Yaskawa INFORM job: DEMO_ROOF_SIDE_0625_3PAINT_14.JBI

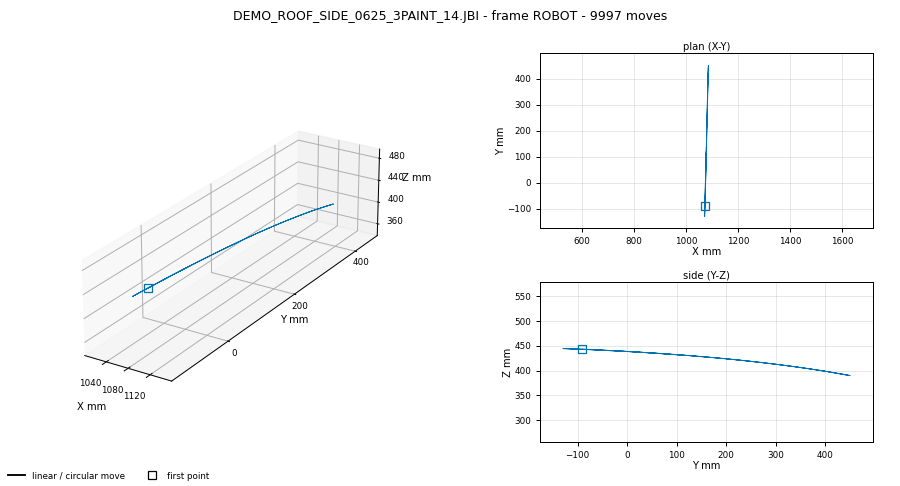
[picture p0: tool path of DEMO_ROOF_SIDE_0625_3PAINT_14.JBI in frame ROBOT, 9997 of 9997 moves have a stored position in this frame; points joined in program order, loops and branches not executed]
/JOB
//NAME DEMO_ROOF_SIDE_0625_3PAINT14
//POS
///NPOS 9997,0,0,0,0,0
///TOOL 0
///USER 0
///POSTYPE ROBOT
///RECTAN
///RCONF 1,0,0,0,0,0,0,0,0,0,0,0,0,0,0,0,0,0,0,0,0,0,0,0
C00000=1074.095,-91.297,443.530,172.904,21.219,153.796
C00001=1074.101,-91.048,443.519,172.905,21.220,153.796
C00002=1074.107,-90.797,443.509,172.907,21.222,153.796
C00003=1074.113,-90.548,443.498,172.908,21.223,153.796
C00004=1074.120,-90.298,443.488,172.910,21.225,153.796
C00005=1074.125,-90.048,443.478,172.911,21.226,153.796
C00006=1074.131,-89.799,443.467,172.913,21.228,153.796
C00007=1074.138,-89.549,443.456,172.914,21.229,153.796
C00008=1074.143,-89.299,443.446,172.916,21.231,153.796
C00009=1074.150,-89.050,443.436,172.917,21.232,153.796
C00010=1074.156,-88.800,443.425,172.919,21.234,153.796
C00011=1074.161,-88.550,443.415,172.921,21.235,153.796
C00012=1074.168,-88.300,443.404,172.922,21.237,153.796
C00013=1074.174,-88.051,443.393,172.924,21.238,153.796
C00014=1074.180,-87.801,443.383,172.925,21.239,153.796
C00015=1074.186,-87.551,443.373,172.927,21.241,153.797
C00016=1074.192,-87.301,443.361,172.928,21.242,153.797
C00017=1074.198,-87.052,443.351,172.930,21.244,153.797
C00018=1074.204,-86.803,443.340,172.931,21.246,153.797
C00019=1074.210,-86.552,443.330,172.933,21.247,153.797
C00020=1074.217,-86.303,443.319,172.934,21.248,153.797
C00021=1074.222,-86.053,443.308,172.936,21.250,153.797
C00022=1074.229,-85.804,443.298,172.937,21.251,153.797
C00023=1074.235,-85.554,443.287,172.939,21.253,153.797
C00024=1074.241,-85.304,443.277,172.941,21.254,153.797
C00025=1074.247,-85.054,443.266,172.942,21.255,153.797
C00026=1074.253,-84.805,443.256,172.943,21.257,153.797
C00027=1074.259,-84.555,443.244,172.945,21.259,153.797
C00028=1074.266,-84.306,443.234,172.947,21.260,153.797
C00029=1074.271,-84.055,443.224,172.948,21.262,153.797
C00030=1074.277,-83.806,443.213,172.950,21.263,153.797
C00031=1074.284,-83.556,443.202,172.951,21.264,153.797
C00032=1074.290,-83.307,443.192,172.953,21.266,153.797
C00033=1074.296,-83.057,443.181,172.954,21.268,153.797
C00034=1074.303,-82.807,443.170,172.956,21.269,153.797
C00035=1074.308,-82.558,443.159,172.957,21.271,153.797
C00036=1074.314,-82.308,443.149,172.959,21.272,153.797
C00037=1074.321,-82.029,443.137,172.961,21.274,153.797
C00038=1074.328,-81.750,443.125,172.962,21.276,153.797
C00039=1074.335,-81.471,443.113,172.964,21.277,153.797
C00040=1074.342,-81.192,443.101,172.965,21.279,153.798
C00041=1074.348,-80.942,443.090,172.967,21.281,153.798
C00042=1074.354,-80.693,443.079,172.968,21.282,153.798
C00043=1074.361,-80.443,443.068,172.971,21.284,153.798
C00044=1074.366,-80.193,443.057,172.972,21.285,153.798
C00045=1074.372,-79.944,443.047,172.974,21.287,153.798
C00046=1074.379,-79.694,443.036,172.975,21.289,153.798
C00047=1074.385,-79.444,443.025,172.977,21.290,153.798
C00048=1074.391,-79.195,443.014,172.978,21.292,153.798
C00049=1074.397,-78.945,443.003,172.980,21.294,153.798
C00050=1074.403,-78.695,442.992,172.981,21.295,153.798
C00051=1074.409,-78.446,442.981,172.983,21.297,153.798
C00052=1074.415,-78.196,442.970,172.984,21.298,153.798
C00053=1074.421,-77.946,442.959,172.986,21.300,153.798
C00054=1074.426,-77.697,442.948,172.987,21.302,153.798
C00055=1074.434,-77.447,442.938,172.989,21.303,153.798
C00056=1074.439,-77.197,442.927,172.990,21.305,153.799
C00057=1074.445,-76.948,442.916,172.992,21.306,153.799
C00058=1074.451,-76.698,442.905,172.993,21.308,153.799
C00059=1074.457,-76.448,442.894,172.995,21.310,153.799
C00060=1074.463,-76.199,442.883,172.996,21.311,153.799
C00061=1074.469,-75.948,442.872,172.997,21.313,153.799
C00062=1074.475,-75.699,442.861,172.999,21.315,153.799
C00063=1074.481,-75.449,442.850,173.001,21.316,153.799
C00064=1074.487,-75.199,442.839,173.002,21.318,153.799
C00065=1074.493,-74.950,442.828,173.003,21.319,153.799
C00066=1074.500,-74.700,442.817,173.005,21.321,153.799
C00067=1074.506,-74.450,442.806,173.006,21.323,153.799
C00068=1074.512,-74.201,442.795,173.008,21.324,153.799
C00069=1074.518,-73.951,442.783,173.009,21.326,153.800
C00070=1074.524,-73.702,442.772,173.011,21.328,153.800
C00071=1074.529,-73.452,442.762,173.012,21.329,153.800
C00072=1074.535,-73.202,442.750,173.014,21.331,153.800
C00073=1074.541,-72.952,442.739,173.015,21.333,153.800
C00074=1074.547,-72.702,442.728,173.016,21.335,153.800
C00075=1074.553,-72.453,442.717,173.019,21.337,153.800
C00076=1074.559,-72.204,442.705,173.020,21.339,153.800
C00077=1074.565,-71.954,442.694,173.022,21.340,153.800
C00078=1074.571,-71.704,442.683,173.023,21.342,153.800
C00079=1074.577,-71.455,442.672,173.025,21.343,153.800
C00080=1074.582,-71.204,442.660,173.026,21.345,153.800
C00081=1074.588,-70.955,442.649,173.027,21.347,153.801
C00082=1074.594,-70.706,442.638,173.029,21.349,153.801
C00083=1074.600,-70.456,442.627,173.030,21.351,153.801
C00084=1074.606,-70.206,442.616,173.032,21.352,153.801
C00085=1074.612,-69.956,442.604,173.033,21.354,153.801
C00086=1074.619,-69.707,442.593,173.035,21.356,153.801
C00087=1074.624,-69.457,442.581,173.036,21.357,153.801
C00088=1074.630,-69.207,442.570,173.037,21.359,153.801
C00089=1074.636,-68.957,442.559,173.039,21.361,153.801
C00090=1074.642,-68.708,442.547,173.040,21.363,153.802
C00091=1074.648,-68.458,442.536,173.042,21.365,153.802
C00092=1074.654,-68.209,442.526,173.043,21.366,153.802
C00093=1074.660,-67.959,442.513,173.045,21.368,153.802
C00094=1074.665,-67.710,442.502,173.046,21.370,153.802
C00095=1074.672,-67.459,442.491,173.048,21.372,153.802
C00096=1074.677,-67.210,442.480,173.050,21.374,153.802
C00097=1074.684,-66.960,442.468,173.051,21.376,153.802
C00098=1074.690,-66.711,442.457,173.053,21.377,153.802
C00099=1074.695,-66.460,442.445,173.054,21.379,153.802
C00100=1074.701,-66.211,442.434,173.055,21.381,153.803
C00101=1074.708,-65.934,442.421,173.057,21.383,153.803
C00102=1074.715,-65.658,442.408,173.058,21.384,153.803
C00103=1074.721,-65.381,442.396,173.060,21.387,153.803
C00104=1074.728,-65.104,442.384,173.062,21.389,153.803
C00105=1074.734,-64.855,442.372,173.063,21.391,153.803
C00106=1074.740,-64.605,442.361,173.065,21.392,153.803
C00107=1074.747,-64.356,442.349,173.066,21.394,153.803
C00108=1074.752,-64.106,442.338,173.067,21.396,153.804
C00109=1074.758,-63.856,442.326,173.069,21.397,153.804
C00110=1074.764,-63.607,442.315,173.070,21.399,153.804
C00111=1074.770,-63.357,442.303,173.072,21.401,153.804
C00112=1074.776,-63.107,442.291,173.073,21.403,153.804
C00113=1074.782,-62.857,442.280,173.075,21.405,153.804
C00114=1074.788,-62.608,442.268,173.077,21.407,153.804
C00115=1074.794,-62.358,442.257,173.078,21.409,153.804
C00116=1074.800,-62.109,442.246,173.080,21.410,153.804
C00117=1074.806,-61.859,442.234,173.081,21.412,153.804
C00118=1074.812,-61.609,442.223,173.082,21.414,153.805
C00119=1074.818,-61.360,442.211,173.084,21.416,153.805
C00120=1074.825,-61.109,442.200,173.085,21.418,153.805
C00121=1074.830,-60.860,442.187,173.087,21.420,153.805
C00122=1074.836,-60.610,442.176,173.088,21.422,153.805
C00123=1074.842,-60.361,442.165,173.090,21.423,153.805
C00124=1074.849,-60.111,442.153,173.091,21.425,153.805
C00125=1074.854,-59.862,442.141,173.092,21.427,153.805
C00126=1074.860,-59.612,442.130,173.094,21.429,153.806
C00127=1074.867,-59.362,442.118,173.095,21.430,153.806
C00128=1074.872,-59.112,442.107,173.097,21.433,153.806
C00129=1074.879,-58.863,442.095,173.099,21.435,153.806
C00130=1074.884,-58.613,442.084,173.100,21.437,153.806
C00131=1074.891,-58.364,442.072,173.102,21.438,153.806
C00132=1074.897,-58.114,442.059,173.103,21.440,153.806
C00133=1074.903,-57.864,442.048,173.104,21.442,153.806
C00134=1074.909,-57.615,442.036,173.106,21.444,153.807
C00135=1074.914,-57.365,442.025,173.107,21.446,153.807
C00136=1074.921,-57.115,442.013,173.109,21.447,153.807
C00137=1074.928,-56.866,442.001,173.110,21.449,153.807
C00138=1074.933,-56.616,441.990,173.111,21.451,153.807
C00139=1074.939,-56.366,441.978,173.113,21.453,153.807
C00140=1074.946,-56.116,441.966,173.114,21.455,153.807
C00141=1074.952,-55.867,441.955,173.117,21.457,153.807
C00142=1074.958,-55.617,441.942,173.118,21.459,153.807
C00143=1074.964,-55.367,441.931,173.119,21.461,153.808
C00144=1074.970,-55.118,441.919,173.121,21.463,153.808
C00145=1074.976,-54.869,441.907,173.122,21.465,153.808
C00146=1074.982,-54.618,441.896,173.124,21.466,153.808
C00147=1074.988,-54.369,441.884,173.125,21.468,153.808
C00148=1074.994,-54.120,441.871,173.126,21.470,153.808
C00149=1075.001,-53.869,441.860,173.128,21.472,153.808
C00150=1075.007,-53.621,441.849,173.129,21.474,153.809
C00151=1075.013,-53.371,441.836,173.130,21.476,153.809
C00152=1075.019,-53.120,441.825,173.132,21.477,153.809
C00153=1075.025,-52.872,441.813,173.134,21.480,153.809
C00154=1075.031,-52.622,441.801,173.135,21.482,153.809
C00155=1075.037,-52.372,441.789,173.137,21.484,153.809
C00156=1075.043,-52.123,441.778,173.138,21.486,153.809
C00157=1075.049,-51.873,441.765,173.140,21.487,153.810
C00158=1075.056,-51.623,441.753,173.141,21.489,153.810
C00159=1075.062,-51.374,441.741,173.142,21.491,153.810
C00160=1075.067,-51.124,441.730,173.144,21.493,153.810
C00161=1075.074,-50.874,441.718,173.145,21.495,153.810
C00162=1075.080,-50.624,441.705,173.147,21.497,153.810
C00163=1075.087,-50.375,441.693,173.148,21.499,153.810
C00164=1075.092,-50.126,441.681,173.150,21.501,153.810
C00165=1075.098,-49.850,441.668,173.152,21.503,153.811
C00166=1075.105,-49.574,441.655,173.153,21.505,153.811
C00167=1075.112,-49.299,441.641,173.154,21.507,153.811
C00168=1075.118,-49.023,441.628,173.156,21.510,153.811
C00169=1075.124,-48.774,441.617,173.158,21.512,153.811
C00170=1075.130,-48.524,441.604,173.159,21.514,153.811
C00171=1075.136,-48.274,441.592,173.160,21.516,153.812
C00172=1075.142,-48.025,441.580,173.162,21.518,153.812
C00173=1075.148,-47.776,441.568,173.163,21.520,153.812
C00174=1075.154,-47.525,441.556,173.164,21.521,153.812
C00175=1075.160,-47.276,441.544,173.166,21.523,153.812
C00176=1075.166,-47.026,441.532,173.168,21.526,153.812
C00177=1075.172,-46.777,441.520,173.169,21.528,153.812
C00178=1075.178,-46.527,441.507,173.171,21.530,153.813
C00179=1075.184,-46.278,441.495,173.172,21.532,153.813
C00180=1075.190,-46.028,441.483,173.173,21.534,153.813
C00181=1075.196,-45.778,441.470,173.175,21.536,153.813
C00182=1075.201,-45.529,441.458,173.176,21.537,153.813
C00183=1075.208,-45.279,441.446,173.178,21.539,153.813
C00184=1075.214,-45.030,441.434,173.179,21.542,153.814
C00185=1075.220,-44.780,441.421,173.181,21.544,153.814
C00186=1075.226,-44.530,441.410,173.182,21.546,153.814
C00187=1075.232,-44.280,441.398,173.184,21.548,153.814
C00188=1075.237,-44.030,441.385,173.185,21.550,153.814
C00189=1075.244,-43.781,441.373,173.186,21.552,153.814
C00190=1075.249,-43.532,441.361,173.188,21.554,153.815
C00191=1075.255,-43.282,441.348,173.189,21.556,153.815
C00192=1075.262,-43.032,441.336,173.190,21.558,153.815
C00193=1075.268,-42.782,441.324,173.192,21.560,153.815
C00194=1075.273,-42.533,441.312,173.193,21.562,153.815
C00195=1075.279,-42.283,441.299,173.195,21.565,153.815
C00196=1075.286,-42.034,441.287,173.197,21.567,153.816
C00197=1075.292,-41.784,441.275,173.198,21.569,153.816
C00198=1075.298,-41.535,441.261,173.199,21.571,153.816
C00199=1075.304,-41.286,441.250,173.201,21.573,153.816
C00200=1075.310,-41.036,441.237,173.202,21.574,153.816
C00201=1075.316,-40.786,441.225,173.203,21.576,153.816
C00202=1075.322,-40.536,441.212,173.205,21.578,153.817
C00203=1075.328,-40.286,441.200,173.206,21.580,153.817
C00204=1075.334,-40.037,441.188,173.208,21.583,153.817
C00205=1075.340,-39.787,441.175,173.209,21.585,153.817
C00206=1075.346,-39.538,441.163,173.211,21.587,153.817
C00207=1075.352,-39.288,441.151,173.212,21.589,153.817
C00208=1075.358,-39.038,441.138,173.214,21.591,153.818
C00209=1075.364,-38.789,441.125,173.215,21.593,153.818
C00210=1075.371,-38.539,441.113,173.216,21.595,153.818
C00211=1075.376,-38.290,441.101,173.217,21.597,153.818
C00212=1075.382,-38.040,441.088,173.219,21.599,153.818
C00213=1075.388,-37.790,441.076,173.221,21.602,153.818
C00214=1075.394,-37.540,441.063,173.222,21.604,153.819
C00215=1075.400,-37.291,441.051,173.224,21.606,153.819
C00216=1075.405,-37.042,441.038,173.225,21.608,153.819
C00217=1075.411,-36.792,441.025,173.226,21.610,153.819
C00218=1075.417,-36.542,441.013,173.228,21.612,153.819
C00219=1075.423,-36.292,441.000,173.229,21.614,153.820
C00220=1075.429,-36.042,440.988,173.230,21.616,153.820
C00221=1075.435,-35.794,440.975,173.232,21.619,153.820
C00222=1075.441,-35.544,440.963,173.234,21.621,153.820
C00223=1075.447,-35.294,440.950,173.235,21.623,153.820
C00224=1075.453,-35.045,440.938,173.236,21.625,153.821
C00225=1075.459,-34.795,440.925,173.238,21.627,153.821
C00226=1075.465,-34.545,440.912,173.239,21.629,153.821
C00227=1075.471,-34.295,440.899,173.240,21.632,153.821
C00228=1075.476,-34.046,440.887,173.242,21.633,153.821
C00229=1075.484,-33.772,440.873,173.244,21.636,153.821
C00230=1075.490,-33.496,440.859,173.245,21.638,153.822
C00231=1075.497,-33.221,440.844,173.246,21.640,153.822
C00232=1075.503,-32.946,440.831,173.248,21.643,153.822
C00233=1075.509,-32.696,440.818,173.250,21.645,153.822
C00234=1075.515,-32.447,440.805,173.251,21.648,153.823
C00235=1075.521,-32.198,440.793,173.252,21.650,153.823
C00236=1075.527,-31.948,440.780,173.254,21.651,153.823
C00237=1075.533,-31.698,440.767,173.255,21.653,153.823
C00238=1075.539,-31.449,440.754,173.257,21.656,153.823
C00239=1075.545,-31.199,440.742,173.258,21.658,153.823
C00240=1075.551,-30.949,440.729,173.260,21.660,153.824
C00241=1075.557,-30.699,440.716,173.261,21.663,153.824
C00242=1075.563,-30.450,440.703,173.262,21.665,153.824
C00243=1075.569,-30.200,440.690,173.264,21.667,153.824
C00244=1075.575,-29.950,440.678,173.265,21.669,153.825
C00245=1075.581,-29.701,440.665,173.266,21.671,153.825
C00246=1075.587,-29.451,440.652,173.269,21.673,153.825
C00247=1075.593,-29.201,440.639,173.270,21.675,153.825
C00248=1075.599,-28.952,440.626,173.271,21.678,153.825
C00249=1075.605,-28.702,440.613,173.272,21.680,153.825
C00250=1075.611,-28.453,440.600,173.274,21.682,153.826
C00251=1075.617,-28.204,440.588,173.275,21.684,153.826
C00252=1075.622,-27.954,440.575,173.276,21.686,153.826
C00253=1075.629,-27.705,440.562,173.278,21.688,153.826
C00254=1075.635,-27.455,440.550,173.280,21.691,153.826
C00255=1075.641,-27.206,440.536,173.281,21.693,153.827
C00256=1075.647,-26.956,440.524,173.282,21.695,153.827
C00257=1075.653,-26.706,440.511,173.284,21.697,153.827
C00258=1075.658,-26.456,440.497,173.285,21.699,153.827
C00259=1075.664,-26.207,440.484,173.286,21.702,153.827
C00260=1075.670,-25.957,440.472,173.288,21.704,153.828
C00261=1075.676,-25.708,440.458,173.290,21.706,153.828
C00262=1075.682,-25.458,440.446,173.291,21.709,153.828
C00263=1075.688,-25.208,440.432,173.292,21.710,153.828
C00264=1075.694,-24.958,440.419,173.294,21.713,153.828
C00265=1075.700,-24.709,440.406,173.295,21.715,153.829
C00266=1075.706,-24.459,440.393,173.296,21.717,153.829
C00267=1075.712,-24.210,440.380,173.297,21.719,153.829
C00268=1075.718,-23.960,440.366,173.300,21.722,153.829
C00269=1075.723,-23.711,440.354,173.301,21.724,153.830
C00270=1075.730,-23.461,440.341,173.302,21.726,153.830
C00271=1075.736,-23.211,440.328,173.303,21.729,153.830
C00272=1075.741,-22.962,440.314,173.305,21.730,153.830
C00273=1075.747,-22.712,440.302,173.306,21.733,153.830
C00274=1075.753,-22.463,440.288,173.307,21.735,153.831
C00275=1075.759,-22.213,440.275,173.308,21.737,153.831
C00276=1075.765,-21.963,440.262,173.311,21.740,153.831
C00277=1075.771,-21.714,440.249,173.312,21.742,153.831
C00278=1075.777,-21.465,440.235,173.313,21.744,153.831
C00279=1075.783,-21.215,440.223,173.315,21.746,153.832
C00280=1075.788,-20.965,440.209,173.316,21.749,153.832
C00281=1075.795,-20.716,440.196,173.317,21.751,153.832
C00282=1075.800,-20.466,440.183,173.318,21.753,153.832
C00283=1075.807,-20.217,440.170,173.321,21.755,153.832
C00284=1075.812,-19.967,440.156,173.322,21.758,153.833
C00285=1075.818,-19.717,440.143,173.323,21.760,153.833
C00286=1075.824,-19.468,440.130,173.324,21.762,153.833
C00287=1075.831,-19.219,440.117,173.326,21.764,153.833
C00288=1075.836,-18.969,440.104,173.327,21.767,153.834
C00289=1075.842,-18.719,440.090,173.328,21.769,153.834
C00290=1075.849,-18.469,440.077,173.330,21.772,153.834
C00291=1075.854,-18.220,440.063,173.332,21.773,153.834
C00292=1075.860,-17.970,440.050,173.333,21.776,153.834
C00293=1075.866,-17.695,440.036,173.334,21.778,153.835
C00294=1075.873,-17.419,440.021,173.336,21.781,153.835
C00295=1075.880,-17.143,440.006,173.337,21.783,153.835
C00296=1075.887,-16.866,439.991,173.339,21.785,153.835
C00297=1075.893,-16.617,439.978,173.341,21.788,153.836
C00298=1075.899,-16.368,439.965,173.342,21.790,153.836
C00299=1075.904,-16.118,439.952,173.343,21.792,153.836
C00300=1075.910,-15.868,439.938,173.345,21.794,153.836
C00301=1075.917,-15.619,439.925,173.346,21.797,153.836
C00302=1075.922,-15.370,439.911,173.347,21.799,153.837
C00303=1075.928,-15.120,439.898,173.349,21.801,153.837
C00304=1075.935,-14.870,439.884,173.351,21.804,153.837
C00305=1075.940,-14.620,439.871,173.352,21.806,153.837
C00306=1075.947,-14.371,439.858,173.353,21.809,153.838
C00307=1075.952,-14.121,439.844,173.354,21.811,153.838
C00308=1075.958,-13.872,439.831,173.356,21.813,153.838
C00309=1075.964,-13.623,439.817,173.357,21.815,153.838
C00310=1075.970,-13.373,439.804,173.359,21.818,153.839
C00311=1075.975,-13.124,439.790,173.360,21.820,153.839
C00312=1075.981,-12.874,439.777,173.362,21.822,153.839
C00313=1075.987,-12.624,439.763,173.363,21.825,153.839
C00314=1075.994,-12.374,439.750,173.364,21.827,153.839
C00315=1075.999,-12.125,439.736,173.365,21.829,153.840
C00316=1076.005,-11.875,439.723,173.367,21.831,153.840
C00317=1076.011,-11.626,439.709,173.369,21.834,153.840
C00318=1076.016,-11.376,439.695,173.370,21.836,153.840
C00319=1076.022,-11.127,439.682,173.371,21.838,153.841
C00320=1076.028,-10.877,439.668,173.373,21.841,153.841
C00321=1076.035,-10.627,439.654,173.374,21.843,153.841
C00322=1076.040,-10.378,439.640,173.375,21.845,153.841
C00323=1076.046,-10.129,439.627,173.377,21.848,153.842
C00324=1076.052,-9.879,439.613,173.379,21.850,153.842
C00325=1076.058,-9.630,439.600,173.380,21.853,153.842
C00326=1076.064,-9.380,439.586,173.381,21.855,153.842
C00327=1076.070,-9.130,439.572,173.382,21.857,153.842
C00328=1076.076,-8.881,439.558,173.383,21.859,153.843
C00329=1076.082,-8.631,439.545,173.386,21.862,153.843
C00330=1076.088,-8.382,439.531,173.387,21.864,153.843
C00331=1076.093,-8.132,439.517,173.388,21.866,153.843
C00332=1076.100,-7.882,439.504,173.389,21.869,153.844
C00333=1076.105,-7.633,439.490,173.391,21.871,153.844
C00334=1076.112,-7.383,439.477,173.392,21.873,153.844
C00335=1076.117,-7.134,439.463,173.393,21.876,153.844
C00336=1076.123,-6.885,439.450,173.395,21.878,153.844
C00337=1076.129,-6.634,439.435,173.397,21.880,153.845
C00338=1076.135,-6.385,439.421,173.398,21.883,153.845
C00339=1076.141,-6.135,439.408,173.399,21.885,153.845
C00340=1076.147,-5.887,439.394,173.400,21.887,153.846
C00341=1076.154,-5.637,439.380,173.402,21.889,153.846
C00342=1076.159,-5.387,439.366,173.404,21.892,153.846
C00343=1076.165,-5.137,439.352,173.405,21.895,153.846
C00344=1076.171,-4.888,439.339,173.406,21.896,153.846
C00345=1076.177,-4.638,439.325,173.408,21.899,153.847
C00346=1076.183,-4.389,439.311,173.409,21.901,153.847
C00347=1076.189,-4.139,439.298,173.410,21.903,153.847
C00348=1076.195,-3.889,439.283,173.412,21.906,153.847
C00349=1076.201,-3.640,439.269,173.414,21.908,153.848
C00350=1076.207,-3.391,439.255,173.415,21.911,153.848
C00351=1076.212,-3.141,439.242,173.416,21.913,153.848
C00352=1076.219,-2.891,439.228,173.417,21.915,153.848
C00353=1076.225,-2.642,439.213,173.419,21.918,153.849
C00354=1076.230,-2.392,439.200,173.421,21.920,153.849
C00355=1076.236,-2.143,439.186,173.422,21.923,153.849
C00356=1076.241,-1.893,439.172,173.423,21.925,153.849
C00357=1076.248,-1.616,439.156,173.424,21.927,153.850
C00358=1076.255,-1.338,439.141,173.426,21.930,153.850
C00359=1076.261,-1.060,439.125,173.428,21.933,153.850
C00360=1076.268,-0.783,439.110,173.429,21.936,153.850
C00361=1076.273,-0.534,439.095,173.431,21.938,153.851
C00362=1076.279,-0.284,439.081,173.432,21.940,153.851
C00363=1076.285,-0.034,439.067,173.433,21.943,153.851
C00364=1076.290,0.215,439.053,173.434,21.945,153.852
C00365=1076.296,0.464,439.038,173.436,21.947,153.852
C00366=1076.302,0.714,439.025,173.438,21.950,153.852
C00367=1076.309,0.964,439.011,173.439,21.953,153.852
C00368=1076.314,1.213,438.996,173.440,21.955,153.853
C00369=1076.320,1.462,438.982,173.442,21.957,153.853
C00370=1076.325,1.712,438.969,173.443,21.960,153.853
C00371=1076.332,1.962,438.954,173.444,21.962,153.853
C00372=1076.337,2.211,438.940,173.446,21.964,153.853
C00373=1076.343,2.461,438.926,173.447,21.967,153.854
C00374=1076.349,2.710,438.911,173.449,21.969,153.854
C00375=1076.355,2.960,438.898,173.450,21.972,153.854
C00376=1076.361,3.209,438.884,173.451,21.974,153.854
C00377=1076.367,3.459,438.869,173.452,21.976,153.855
C00378=1076.373,3.709,438.855,173.454,21.979,153.855
C00379=1076.378,3.957,438.840,173.456,21.981,153.855
C00380=1076.384,4.208,438.826,173.457,21.983,153.855
C00381=1076.390,4.457,438.812,173.458,21.986,153.856
C00382=1076.396,4.706,438.798,173.459,21.988,153.856
C00383=1076.402,4.957,438.784,173.461,21.991,153.856
C00384=1076.408,5.206,438.769,173.463,21.993,153.856
C00385=1076.413,5.455,438.755,173.464,21.996,153.857
C00386=1076.419,5.705,438.740,173.465,21.998,153.857
C00387=1076.425,5.954,438.726,173.466,22.001,153.857
C00388=1076.431,6.203,438.712,173.468,22.002,153.857
C00389=1076.437,6.453,438.698,173.470,22.005,153.858
C00390=1076.443,6.702,438.684,173.471,22.008,153.858
C00391=1076.449,6.952,438.669,173.472,22.010,153.858
C00392=1076.455,7.201,438.655,173.474,22.012,153.858
C00393=1076.461,7.451,438.641,173.475,22.015,153.859
C00394=1076.467,7.701,438.626,173.476,22.017,153.859
C00395=1076.472,7.950,438.612,173.478,22.020,153.859
C00396=1076.479,8.200,438.597,173.480,22.022,153.859
C00397=1076.484,8.449,438.583,173.481,22.024,153.860
C00398=1076.490,8.698,438.569,173.482,22.027,153.860
C00399=1076.496,8.949,438.554,173.483,22.029,153.860
C00400=1076.502,9.198,438.540,173.485,22.032,153.860
C00401=1076.508,9.448,438.526,173.487,22.034,153.861
C00402=1076.514,9.697,438.511,173.488,22.037,153.861
C00403=1076.520,9.947,438.496,173.489,22.039,153.861
C00404=1076.526,10.196,438.482,173.490,22.041,153.862
C00405=1076.532,10.446,438.467,173.492,22.043,153.862
C00406=1076.537,10.695,438.453,173.494,22.046,153.862
C00407=1076.543,10.944,438.439,173.495,22.048,153.862
C00408=1076.550,11.194,438.424,173.496,22.051,153.862
C00409=1076.555,11.444,438.410,173.497,22.053,153.863
C00410=1076.562,11.693,438.395,173.499,22.056,153.863
C00411=1076.567,11.942,438.380,173.501,22.058,153.863
C00412=1076.573,12.192,438.366,173.502,22.060,153.863
C00413=1076.579,12.441,438.352,173.503,22.063,153.864
C00414=1076.586,12.691,438.337,173.505,22.065,153.864
C00415=1076.591,12.941,438.323,173.506,22.067,153.864
C00416=1076.597,13.190,438.308,173.508,22.070,153.864
C00417=1076.603,13.439,438.293,173.509,22.073,153.865
C00418=1076.609,13.690,438.279,173.510,22.075,153.865
C00419=1076.615,13.938,438.265,173.512,22.077,153.865
C00420=1076.621,14.188,438.250,173.513,22.079,153.866
C00421=1076.628,14.468,438.234,173.515,22.082,153.866
C00422=1076.635,14.747,438.217,173.516,22.085,153.866
C00423=1076.641,15.026,438.201,173.518,22.088,153.866
C00424=1076.647,15.306,438.184,173.519,22.090,153.867
C00425=1076.653,15.556,438.169,173.521,22.093,153.867
C00426=1076.659,15.805,438.155,173.522,22.095,153.867
C00427=1076.665,16.054,438.140,173.524,22.098,153.867
C00428=1076.671,16.304,438.125,173.525,22.100,153.868
C00429=1076.677,16.554,438.110,173.526,22.102,153.868
C00430=1076.682,16.803,438.096,173.528,22.105,153.868
C00431=1076.689,17.053,438.081,173.529,22.107,153.869
C00432=1076.695,17.302,438.066,173.531,22.110,153.869
C00433=1076.700,17.552,438.051,173.532,22.113,153.869
C00434=1076.706,17.801,438.037,173.534,22.114,153.869
C00435=1076.712,18.051,438.022,173.535,22.117,153.870
C00436=1076.718,18.300,438.007,173.536,22.119,153.870
C00437=1076.723,18.550,437.992,173.538,22.122,153.870
C00438=1076.729,18.799,437.977,173.539,22.125,153.870
C00439=1076.736,19.048,437.962,173.540,22.127,153.871
C00440=1076.741,19.297,437.948,173.542,22.129,153.871
C00441=1076.747,19.548,437.933,173.543,22.132,153.871
C00442=1076.753,19.797,437.918,173.545,22.134,153.871
C00443=1076.759,20.046,437.903,173.546,22.137,153.872
C00444=1076.765,20.296,437.888,173.548,22.139,153.872
C00445=1076.770,20.545,437.873,173.549,22.141,153.872
C00446=1076.777,20.795,437.858,173.550,22.144,153.872
C00447=1076.783,21.044,437.844,173.552,22.147,153.873
C00448=1076.788,21.294,437.828,173.553,22.149,153.873
C00449=1076.794,21.543,437.814,173.555,22.151,153.873
C00450=1076.800,21.793,437.798,173.556,22.154,153.874
C00451=1076.805,22.042,437.784,173.557,22.156,153.874
C00452=1076.812,22.291,437.769,173.559,22.159,153.874
C00453=1076.817,22.541,437.753,173.560,22.161,153.874
C00454=1076.823,22.790,437.738,173.562,22.164,153.875
C00455=1076.830,23.040,437.723,173.563,22.166,153.875
C00456=1076.835,23.289,437.708,173.564,22.169,153.875
C00457=1076.841,23.539,437.693,173.566,22.171,153.875
C00458=1076.847,23.789,437.678,173.568,22.173,153.876
C00459=1076.852,24.038,437.663,173.569,22.176,153.876
C00460=1076.859,24.288,437.648,173.570,22.178,153.876
C00461=1076.864,24.537,437.633,173.571,22.181,153.876
C00462=1076.870,24.786,437.618,173.573,22.184,153.877
C00463=1076.876,25.036,437.603,173.574,22.186,153.877
C00464=1076.882,25.285,437.588,173.576,22.188,153.877
C00465=1076.888,25.535,437.573,173.577,22.190,153.877
C00466=1076.893,25.784,437.558,173.578,22.193,153.878
C00467=1076.899,26.034,437.543,173.580,22.196,153.878
C00468=1076.905,26.284,437.527,173.582,22.198,153.878
C00469=1076.911,26.533,437.513,173.583,22.200,153.878
C00470=1076.917,26.783,437.498,173.584,22.202,153.879
C00471=1076.923,27.032,437.482,173.585,22.205,153.879
C00472=1076.929,27.281,437.467,173.587,22.208,153.879
C00473=1076.935,27.531,437.452,173.589,22.210,153.880
C00474=1076.940,27.780,437.437,173.590,22.213,153.880
C00475=1076.946,28.030,437.421,173.591,22.215,153.880
C00476=1076.952,28.279,437.406,173.593,22.218,153.880
C00477=1076.958,28.529,437.391,173.595,22.220,153.881
C00478=1076.964,28.778,437.376,173.596,22.222,153.881
C00479=1076.970,29.028,437.360,173.597,22.225,153.881
C00480=1076.976,29.277,437.346,173.598,22.227,153.881
C00481=1076.981,29.527,437.330,173.600,22.230,153.882
C00482=1076.987,29.777,437.314,173.601,22.233,153.882
C00483=1076.993,30.025,437.299,173.603,22.235,153.882
C00484=1076.999,30.275,437.284,173.604,22.237,153.882
C00485=1077.005,30.556,437.267,173.606,22.240,153.883
C00486=1077.012,30.836,437.250,173.607,22.243,153.883
C00487=1077.018,31.117,437.232,173.609,22.246,153.883
C00488=1077.025,31.399,437.215,173.611,22.248,153.884
C00489=1077.031,31.647,437.199,173.612,22.251,153.884
C00490=1077.036,31.897,437.184,173.614,22.253,153.884
C00491=1077.043,32.147,437.169,173.615,22.256,153.885
C00492=1077.048,32.396,437.153,173.616,22.258,153.885
C00493=1077.054,32.624,437.139,173.618,22.260,153.885
C00494=1077.059,32.853,437.125,173.619,22.263,153.885
C00495=1077.064,33.081,437.110,173.620,22.265,153.886
C00496=1077.069,33.310,437.097,173.621,22.267,153.886
C00497=1077.074,33.539,437.083,173.623,22.270,153.886
C00498=1077.080,33.767,437.069,173.624,22.272,153.886
C00499=1077.085,33.995,437.054,173.625,22.274,153.886
C00500=1077.090,34.224,437.040,173.626,22.276,153.887
C00501=1077.097,34.473,437.025,173.629,22.279,153.887
C00502=1077.103,34.723,437.009,173.630,22.281,153.887
C00503=1077.108,34.973,436.993,173.631,22.284,153.888
C00504=1077.114,35.222,436.978,173.632,22.286,153.888
C00505=1077.120,35.471,436.962,173.634,22.289,153.888
C00506=1077.126,35.721,436.947,173.636,22.291,153.888
C00507=1077.132,35.971,436.932,173.637,22.294,153.889
C00508=1077.138,36.219,436.916,173.638,22.296,153.889
C00509=1077.143,36.469,436.900,173.640,22.298,153.889
C00510=1077.150,36.718,436.885,173.642,22.301,153.889
C00511=1077.156,36.968,436.869,173.643,22.303,153.890
C00512=1077.161,37.217,436.854,173.644,22.306,153.890
C00513=1077.167,37.466,436.838,173.645,22.308,153.890
C00514=1077.173,37.716,436.823,173.647,22.311,153.890
C00515=1077.179,37.966,436.806,173.649,22.313,153.891
C00516=1077.184,38.215,436.791,173.650,22.316,153.891
C00517=1077.191,38.464,436.776,173.651,22.318,153.891
C00518=1077.196,38.714,436.760,173.653,22.321,153.891
C00519=1077.202,38.963,436.744,173.654,22.323,153.892
C00520=1077.207,39.213,436.729,173.656,22.326,153.892
C00521=1077.213,39.462,436.712,173.657,22.328,153.892
C00522=1077.219,39.712,436.697,173.658,22.331,153.893
C00523=1077.226,39.961,436.681,173.660,22.333,153.893
C00524=1077.231,40.211,436.666,173.661,22.336,153.893
C00525=1077.237,40.460,436.650,173.663,22.338,153.893
C00526=1077.242,40.710,436.634,173.664,22.340,153.894
C00527=1077.248,40.959,436.618,173.666,22.343,153.894
C00528=1077.254,41.208,436.602,173.667,22.346,153.894
C00529=1077.260,41.458,436.586,173.669,22.348,153.895
C00530=1077.265,41.707,436.570,173.670,22.350,153.895
C00531=1077.271,41.957,436.555,173.672,22.353,153.895
C00532=1077.277,42.206,436.539,173.673,22.356,153.895
C00533=1077.283,42.456,436.523,173.675,22.358,153.896
C00534=1077.289,42.705,436.507,173.676,22.360,153.896
C00535=1077.294,42.954,436.491,173.678,22.363,153.896
C00536=1077.300,43.204,436.476,173.679,22.365,153.896
C00537=1077.306,43.453,436.459,173.680,22.368,153.897
C00538=1077.312,43.703,436.443,173.682,22.370,153.897
C00539=1077.318,43.953,436.428,173.684,22.373,153.897
C00540=1077.323,44.202,436.411,173.685,22.376,153.898
C00541=1077.329,44.451,436.396,173.686,22.378,153.898
C00542=1077.334,44.701,436.380,173.687,22.380,153.898
C00543=1077.340,44.950,436.364,173.689,22.383,153.898
C00544=1077.346,45.199,436.347,173.691,22.386,153.899
C00545=1077.351,45.448,436.332,173.692,22.388,153.899
C00546=1077.357,45.698,436.316,173.693,22.390,153.899
C00547=1077.363,45.947,436.300,173.695,22.393,153.899
C00548=1077.369,46.197,436.284,173.697,22.395,153.900
C00549=1077.376,46.520,436.263,173.698,22.399,153.900
C00550=1077.384,46.843,436.242,173.700,22.402,153.900
C00551=1077.391,47.165,436.222,173.702,22.406,153.901
C00552=1077.398,47.488,436.200,173.703,22.409,153.901
C00553=1077.404,47.737,436.184,173.706,22.411,153.901
C00554=1077.410,47.987,436.169,173.707,22.413,153.902
C00555=1077.416,48.237,436.152,173.708,22.416,153.902
C00556=1077.422,48.486,436.136,173.709,22.418,153.902
C00557=1077.428,48.735,436.120,173.711,22.421,153.903
C00558=1077.433,48.984,436.104,173.713,22.423,153.903
C00559=1077.438,49.234,436.088,173.714,22.426,153.903
C00560=1077.444,49.484,436.071,173.715,22.428,153.903
C00561=1077.450,49.733,436.055,173.717,22.431,153.904
C00562=1077.456,49.982,436.039,173.718,22.434,153.904
C00563=1077.462,50.232,436.023,173.720,22.436,153.904
C00564=1077.468,50.481,436.006,173.721,22.438,153.905
C00565=1077.473,50.731,435.991,173.723,22.441,153.905
C00566=1077.478,50.981,435.974,173.724,22.443,153.905
C00567=1077.484,51.230,435.958,173.726,22.446,153.905
C00568=1077.490,51.479,435.942,173.728,22.448,153.906
C00569=1077.496,51.728,435.926,173.729,22.451,153.906
C00570=1077.502,51.977,435.909,173.730,22.453,153.906
C00571=1077.508,52.227,435.893,173.731,22.456,153.906
C00572=1077.514,52.476,435.877,173.733,22.459,153.907
C00573=1077.519,52.726,435.860,173.735,22.461,153.907
C00574=1077.525,52.975,435.844,173.736,22.463,153.907
C00575=1077.531,53.224,435.827,173.737,22.465,153.907
C00576=1077.537,53.474,435.811,173.739,22.468,153.908
C00577=1077.543,53.723,435.795,173.741,22.471,153.908
C00578=1077.547,53.973,435.779,173.742,22.473,153.908
C00579=1077.553,54.223,435.763,173.743,22.476,153.909
C00580=1077.559,54.472,435.746,173.745,22.478,153.909
C00581=1077.565,54.721,435.730,173.747,22.480,153.909
C00582=1077.571,54.971,435.714,173.748,22.483,153.909
C00583=1077.577,55.220,435.698,173.750,22.486,153.910
C00584=1077.583,55.469,435.680,173.751,22.488,153.910
C00585=1077.589,55.719,435.664,173.752,22.490,153.910
C00586=1077.595,55.968,435.647,173.754,22.493,153.910
C00587=1077.601,56.217,435.631,173.756,22.495,153.911
C00588=1077.606,56.467,435.614,173.757,22.498,153.911
C00589=1077.612,56.716,435.598,173.758,22.500,153.911
C00590=1077.618,56.966,435.582,173.760,22.503,153.911
C00591=1077.624,57.215,435.566,173.762,22.505,153.912
C00592=1077.630,57.464,435.549,173.763,22.508,153.912
C00593=1077.635,57.714,435.533,173.764,22.510,153.912
C00594=1077.641,57.963,435.516,173.767,22.513,153.912
C00595=1077.647,58.213,435.500,173.768,22.515,153.913
C00596=1077.653,58.462,435.484,173.769,22.517,153.913
C00597=1077.658,58.711,435.466,173.770,22.520,153.913
C00598=1077.664,58.960,435.450,173.773,22.522,153.913
C00599=1077.670,59.210,435.434,173.774,22.525,153.914
C00600=1077.676,59.459,435.417,173.775,22.527,153.914
C00601=1077.681,59.709,435.401,173.776,22.529,153.914
C00602=1077.688,59.959,435.384,173.778,22.532,153.915
C00603=1077.694,60.208,435.367,173.780,22.534,153.915
C00604=1077.700,60.457,435.351,173.781,22.537,153.915
C00605=1077.705,60.707,435.334,173.783,22.539,153.915
C00606=1077.711,60.956,435.318,173.784,22.542,153.916
C00607=1077.717,61.205,435.301,173.786,22.544,153.916
C00608=1077.723,61.454,435.284,173.787,22.546,153.916
C00609=1077.729,61.704,435.268,173.789,22.549,153.916
C00610=1077.735,61.953,435.251,173.790,22.551,153.917
C00611=1077.741,62.203,435.235,173.792,22.554,153.917
C00612=1077.746,62.453,435.218,173.794,22.556,153.917
C00613=1077.753,62.732,435.199,173.795,22.559,153.917
C00614=1077.760,63.013,435.181,173.797,22.561,153.918
C00615=1077.766,63.293,435.161,173.798,22.564,153.918
C00616=1077.773,63.574,435.143,173.800,22.567,153.918
C00617=1077.779,63.824,435.127,173.802,22.569,153.918
C00618=1077.785,64.073,435.109,173.803,22.572,153.919
C00619=1077.791,64.323,435.092,173.805,22.574,153.919
C00620=1077.797,64.572,435.076,173.806,22.577,153.919
C00621=1077.803,64.821,435.059,173.808,22.579,153.919
C00622=1077.809,65.071,435.042,173.810,22.582,153.920
C00623=1077.814,65.320,435.025,173.811,22.584,153.920
C00624=1077.820,65.569,435.008,173.812,22.586,153.920
C00625=1077.825,65.819,434.992,173.814,22.589,153.921
C00626=1077.831,66.068,434.975,173.816,22.592,153.921
C00627=1077.837,66.318,434.957,173.817,22.594,153.921
C00628=1077.843,66.567,434.941,173.818,22.596,153.921
C00629=1077.848,66.817,434.924,173.820,22.599,153.922
C00630=1077.855,67.066,434.907,173.822,22.601,153.922
C00631=1077.860,67.315,434.890,173.823,22.604,153.922
C00632=1077.866,67.564,434.873,173.825,22.606,153.922
C00633=1077.871,67.814,434.857,173.826,22.608,153.923
C00634=1077.878,68.063,434.839,173.828,22.611,153.923
C00635=1077.883,68.313,434.822,173.830,22.614,153.923
C00636=1077.889,68.562,434.806,173.831,22.616,153.923
C00637=1077.895,68.811,434.789,173.833,22.618,153.924
C00638=1077.900,69.061,434.772,173.834,22.620,153.924
C00639=1077.906,69.309,434.755,173.836,22.623,153.924
C00640=1077.912,69.560,434.738,173.837,22.626,153.924
C00641=1077.918,69.809,434.720,173.838,22.628,153.925
C00642=1077.924,70.058,434.704,173.841,22.630,153.925
C00643=1077.929,70.307,434.686,173.842,22.633,153.925
C00644=1077.935,70.557,434.670,173.843,22.635,153.925
C00645=1077.941,70.806,434.652,173.845,22.638,153.926
C00646=1077.946,71.056,434.635,173.846,22.641,153.926
C00647=1077.953,71.305,434.618,173.848,22.643,153.926
C00648=1077.958,71.554,434.601,173.850,22.645,153.926
C00649=1077.963,71.803,434.584,173.851,22.648,153.927
C00650=1077.970,72.052,434.567,173.853,22.650,153.927
C00651=1077.976,72.302,434.550,173.854,22.653,153.927
C00652=1077.981,72.552,434.532,173.856,22.655,153.928
C00653=1077.986,72.801,434.515,173.857,22.657,153.928
C00654=1077.993,73.050,434.498,173.859,22.660,153.928
C00655=1077.998,73.299,434.481,173.861,22.662,153.928
C00656=1078.004,73.549,434.463,173.862,22.665,153.929
C00657=1078.010,73.798,434.446,173.863,22.667,153.929
C00658=1078.016,74.047,434.429,173.865,22.670,153.929
C00659=1078.021,74.297,434.412,173.867,22.672,153.929
C00660=1078.027,74.546,434.394,173.868,22.674,153.930
C00661=1078.033,74.795,434.377,173.870,22.677,153.930
C00662=1078.038,75.045,434.360,173.871,22.679,153.930
C00663=1078.044,75.294,434.343,173.873,22.682,153.930
C00664=1078.050,75.544,434.325,173.875,22.684,153.931
C00665=1078.056,75.793,434.308,173.876,22.687,153.931
C00666=1078.062,76.042,434.291,173.877,22.689,153.931
C00667=1078.067,76.291,434.273,173.880,22.692,153.931
C00668=1078.073,76.541,434.256,173.881,22.694,153.932
C00669=1078.079,76.790,434.239,173.882,22.696,153.932
C00670=1078.085,77.039,434.222,173.884,22.699,153.932
C00671=1078.090,77.288,434.204,173.886,22.701,153.932
C00672=1078.096,77.539,434.187,173.887,22.704,153.933
C00673=1078.102,77.788,434.169,173.889,22.706,153.933
C00674=1078.108,78.036,434.152,173.890,22.709,153.933
C00675=1078.114,78.286,434.134,173.892,22.711,153.933
C00676=1078.119,78.536,434.117,173.894,22.714,153.934
C00677=1078.125,78.817,434.097,173.895,22.716,153.934
C00678=1078.132,79.097,434.078,173.897,22.719,153.934
C00679=1078.138,79.377,434.058,173.898,22.721,153.934
C00680=1078.145,79.658,434.039,173.900,22.725,153.935
C00681=1078.150,79.907,434.021,173.902,22.726,153.935
C00682=1078.156,80.156,434.004,173.904,22.729,153.935
C00683=1078.162,80.406,433.986,173.905,22.732,153.936
C00684=1078.168,80.655,433.968,173.906,22.734,153.936
C00685=1078.173,80.904,433.951,173.909,22.737,153.936
C00686=1078.179,81.154,433.933,173.910,22.739,153.936
C00687=1078.184,81.403,433.916,173.911,22.741,153.937
C00688=1078.190,81.652,433.898,173.913,22.744,153.937
C00689=1078.195,81.901,433.881,173.915,22.746,153.937
C00690=1078.202,82.151,433.863,173.916,22.749,153.937
C00691=1078.207,82.400,433.845,173.918,22.751,153.938
C00692=1078.213,82.649,433.828,173.919,22.754,153.938
C00693=1078.219,82.899,433.810,173.922,22.756,153.938
C00694=1078.224,83.148,433.792,173.923,22.759,153.938
C00695=1078.230,83.397,433.775,173.924,22.761,153.939
C00696=1078.236,83.647,433.757,173.926,22.764,153.939
C00697=1078.241,83.896,433.739,173.928,22.766,153.939
C00698=1078.247,84.145,433.722,173.929,22.768,153.939
C00699=1078.253,84.395,433.704,173.931,22.771,153.940
C00700=1078.259,84.644,433.686,173.932,22.773,153.940
C00701=1078.265,84.893,433.668,173.934,22.775,153.940
C00702=1078.270,85.142,433.651,173.936,22.778,153.940
C00703=1078.276,85.391,433.633,173.937,22.780,153.941
C00704=1078.282,85.641,433.615,173.939,22.783,153.941
C00705=1078.287,85.890,433.598,173.941,22.785,153.941
C00706=1078.293,86.140,433.580,173.942,22.787,153.941
C00707=1078.299,86.389,433.562,173.943,22.790,153.942
C00708=1078.305,86.638,433.544,173.945,22.793,153.942
C00709=1078.311,86.888,433.527,173.947,22.794,153.942
C00710=1078.316,87.137,433.509,173.949,22.797,153.942
C00711=1078.322,87.387,433.491,173.950,22.800,153.943
C00712=1078.328,87.636,433.473,173.952,22.802,153.943
C00713=1078.333,87.885,433.456,173.954,22.804,153.943
C00714=1078.339,88.135,433.437,173.955,22.807,153.943
C00715=1078.345,88.383,433.419,173.957,22.809,153.943
C00716=1078.351,88.633,433.401,173.959,22.811,153.944
C00717=1078.356,88.882,433.384,173.960,22.814,153.944
C00718=1078.362,89.132,433.366,173.961,22.816,153.944
C00719=1078.368,89.381,433.348,173.964,22.819,153.944
C00720=1078.374,89.630,433.330,173.965,22.821,153.945
C00721=1078.379,89.879,433.313,173.967,22.823,153.945
C00722=1078.386,90.129,433.294,173.968,22.826,153.945
C00723=1078.391,90.378,433.276,173.970,22.828,153.945
C00724=1078.398,90.627,433.258,173.972,22.830,153.946
C00725=1078.403,90.876,433.241,173.973,22.833,153.946
C00726=1078.408,91.126,433.223,173.974,22.835,153.946
C00727=1078.414,91.375,433.204,173.977,22.837,153.946
C00728=1078.420,91.624,433.186,173.978,22.840,153.947
C00729=1078.425,91.874,433.168,173.980,22.843,153.947
C00730=1078.431,92.123,433.150,173.981,22.845,153.947
C00731=1078.437,92.372,433.132,173.983,22.847,153.947
C00732=1078.443,92.621,433.114,173.985,22.850,153.948
C00733=1078.448,92.871,433.096,173.986,22.852,153.948
C00734=1078.454,93.120,433.078,173.988,22.854,153.948
C00735=1078.459,93.369,433.060,173.990,22.857,153.948
C00736=1078.465,93.619,433.041,173.991,22.859,153.949
C00737=1078.470,93.868,433.024,173.993,22.862,153.949
C00738=1078.477,94.117,433.005,173.995,22.864,153.949
C00739=1078.482,94.366,432.987,173.996,22.866,153.949
C00740=1078.488,94.616,432.969,173.998,22.869,153.949
C00741=1078.494,94.896,432.948,173.999,22.871,153.950
C00742=1078.500,95.177,432.928,174.001,22.874,153.950
C00743=1078.507,95.457,432.907,174.004,22.877,153.950
C00744=1078.513,95.738,432.887,174.006,22.880,153.951
C00745=1078.520,95.987,432.869,174.007,22.882,153.951
C00746=1078.524,96.237,432.851,174.008,22.884,153.951
C00747=1078.531,96.486,432.832,174.011,22.887,153.951
C00748=1078.536,96.735,432.814,174.012,22.889,153.952
C00749=1078.542,96.984,432.795,174.013,22.891,153.952
C00750=1078.547,97.233,432.778,174.016,22.894,153.952
C00751=1078.554,97.483,432.760,174.017,22.896,153.952
C00752=1078.559,97.732,432.741,174.019,22.899,153.953
C00753=1078.565,97.982,432.723,174.020,22.901,153.953
C00754=1078.571,98.231,432.704,174.022,22.903,153.953
C00755=1078.576,98.480,432.686,174.024,22.905,153.953
C00756=1078.582,98.729,432.667,174.025,22.908,153.953
C00757=1078.587,98.979,432.649,174.027,22.911,153.954
C00758=1078.594,99.228,432.631,174.029,22.913,153.954
C00759=1078.599,99.477,432.613,174.030,22.915,153.954
C00760=1078.605,99.726,432.594,174.032,22.917,153.954
C00761=1078.611,99.976,432.576,174.034,22.920,153.955
C00762=1078.617,100.224,432.558,174.036,22.922,153.955
C00763=1078.622,100.474,432.539,174.037,22.924,153.955
C00764=1078.628,100.723,432.521,174.039,22.927,153.955
C00765=1078.633,100.973,432.502,174.041,22.929,153.955
C00766=1078.640,101.222,432.484,174.042,22.931,153.956
C00767=1078.645,101.471,432.465,174.044,22.934,153.956
C00768=1078.651,101.720,432.447,174.046,22.936,153.956
C00769=1078.656,101.969,432.428,174.048,22.939,153.956
C00770=1078.662,102.219,432.410,174.049,22.941,153.957
C00771=1078.668,102.468,432.391,174.051,22.943,153.957
C00772=1078.674,102.717,432.372,174.053,22.946,153.957
C00773=1078.679,102.967,432.354,174.054,22.948,153.957
C00774=1078.684,103.216,432.335,174.056,22.951,153.958
C00775=1078.690,103.465,432.317,174.058,22.953,153.958
C00776=1078.695,103.714,432.298,174.060,22.955,153.958
C00777=1078.702,103.963,432.280,174.061,22.958,153.958
C00778=1078.707,104.213,432.261,174.062,22.960,153.959
C00779=1078.712,104.462,432.242,174.065,22.962,153.959
C00780=1078.719,104.711,432.223,174.066,22.965,153.959
C00781=1078.724,104.960,432.204,174.068,22.967,153.959
C00782=1078.730,105.209,432.187,174.070,22.970,153.960
C00783=1078.736,105.459,432.167,174.071,22.972,153.960
C00784=1078.741,105.708,432.148,174.073,22.974,153.960
C00785=1078.747,105.957,432.131,174.074,22.977,153.960
C00786=1078.752,106.207,432.111,174.077,22.979,153.960
C00787=1078.758,106.456,432.092,174.078,22.981,153.961
C00788=1078.764,106.705,432.074,174.080,22.984,153.961
C00789=1078.769,106.955,432.055,174.082,22.986,153.961
C00790=1078.775,107.203,432.037,174.084,22.989,153.961
C00791=1078.781,107.453,432.018,174.085,22.991,153.962
C00792=1078.787,107.702,431.999,174.086,22.993,153.962
C00793=1078.793,107.951,431.980,174.089,22.995,153.962
C00794=1078.798,108.201,431.962,174.090,22.998,153.962
C00795=1078.803,108.450,431.942,174.092,23.000,153.962
C00796=1078.810,108.699,431.924,174.094,23.002,153.963
C00797=1078.815,108.948,431.905,174.096,23.005,153.963
C00798=1078.821,109.197,431.886,174.097,23.007,153.963
C00799=1078.827,109.446,431.867,174.100,23.009,153.963
C00800=1078.832,109.696,431.849,174.101,23.012,153.964
C00801=1078.838,109.945,431.830,174.102,23.014,153.964
C00802=1078.844,110.194,431.811,174.104,23.016,153.964
C00803=1078.850,110.444,431.792,174.106,23.018,153.964
C00804=1078.855,110.692,431.773,174.108,23.021,153.964
C00805=1078.862,110.973,431.752,174.110,23.024,153.965
C00806=1078.868,111.254,431.730,174.112,23.026,153.965
C00807=1078.875,111.535,431.709,174.114,23.029,153.965
C00808=1078.881,111.815,431.687,174.116,23.031,153.965
C00809=1078.886,112.065,431.669,174.117,23.034,153.966
C00810=1078.893,112.314,431.650,174.120,23.036,153.966
C00811=1078.898,112.563,431.631,174.121,23.038,153.966
C00812=1078.904,112.812,431.612,174.123,23.041,153.966
C00813=1078.909,113.062,431.593,174.124,23.043,153.967
C00814=1078.915,113.311,431.573,174.127,23.045,153.967
C00815=1078.921,113.559,431.555,174.128,23.048,153.967
C00816=1078.926,113.809,431.536,174.130,23.050,153.967
C00817=1078.932,114.058,431.517,174.132,23.052,153.967
C00818=1078.938,114.308,431.497,174.133,23.054,153.968
C00819=1078.943,114.557,431.478,174.135,23.057,153.968
C00820=1078.949,114.805,431.459,174.137,23.059,153.968
C00821=1078.955,115.055,431.439,174.139,23.062,153.968
C00822=1078.960,115.304,431.420,174.140,23.064,153.969
C00823=1078.965,115.553,431.401,174.142,23.066,153.969
C00824=1078.971,115.802,431.382,174.144,23.069,153.969
C00825=1078.977,116.052,431.363,174.146,23.071,153.969
C00826=1078.982,116.301,431.344,174.147,23.073,153.969
C00827=1078.987,116.550,431.325,174.150,23.076,153.970
C00828=1078.993,116.799,431.305,174.151,23.078,153.970
C00829=1078.999,117.049,431.286,174.153,23.081,153.970
C00830=1079.005,117.298,431.267,174.155,23.083,153.970
C00831=1079.010,117.546,431.247,174.157,23.086,153.971
C00832=1079.016,117.796,431.228,174.158,23.087,153.971
C00833=1079.021,118.045,431.209,174.160,23.090,153.971
C00834=1079.027,118.295,431.190,174.162,23.092,153.971
C00835=1079.033,118.544,431.170,174.164,23.095,153.971
C00836=1079.038,118.792,431.151,174.165,23.097,153.972
C00837=1079.044,119.042,431.132,174.168,23.099,153.972
C00838=1079.049,119.291,431.112,174.169,23.101,153.972
C00839=1079.055,119.541,431.093,174.170,23.104,153.972
C00840=1079.061,119.790,431.074,174.173,23.106,153.972
C00841=1079.067,120.039,431.054,174.174,23.108,153.973
C00842=1079.071,120.288,431.034,174.176,23.111,153.973
C00843=1079.077,120.537,431.015,174.178,23.113,153.973
C00844=1079.083,120.787,430.996,174.180,23.115,153.973
C00845=1079.089,121.035,430.976,174.181,23.118,153.974
C00846=1079.094,121.285,430.957,174.183,23.120,153.974
C00847=1079.100,121.534,430.937,174.185,23.122,153.974
C00848=1079.105,121.782,430.918,174.187,23.125,153.974
C00849=1079.111,122.032,430.899,174.188,23.127,153.974
C00850=1079.117,122.281,430.879,174.191,23.129,153.975
C00851=1079.123,122.530,430.859,174.192,23.132,153.975
C00852=1079.128,122.780,430.840,174.194,23.134,153.975
C00853=1079.134,123.029,430.821,174.196,23.136,153.975
C00854=1079.139,123.278,430.800,174.198,23.139,153.975
C00855=1079.145,123.528,430.781,174.200,23.141,153.976
C00856=1079.151,123.777,430.762,174.202,23.143,153.976
C00857=1079.156,124.025,430.742,174.204,23.145,153.976
C00858=1079.162,124.275,430.723,174.205,23.148,153.976
C00859=1079.167,124.524,430.704,174.208,23.150,153.976
C00860=1079.173,124.773,430.684,174.209,23.153,153.977
C00861=1079.179,125.022,430.665,174.211,23.155,153.977
C00862=1079.184,125.271,430.644,174.213,23.157,153.977
C00863=1079.190,125.521,430.625,174.215,23.159,153.977
C00864=1079.196,125.770,430.605,174.216,23.161,153.977
C00865=1079.202,126.019,430.586,174.219,23.164,153.978
C00866=1079.208,126.268,430.566,174.220,23.166,153.978
C00867=1079.213,126.517,430.546,174.222,23.168,153.978
C00868=1079.219,126.766,430.526,174.223,23.171,153.978
C00869=1079.226,127.047,430.505,174.226,23.173,153.978
C00870=1079.231,127.328,430.482,174.228,23.176,153.979
C00871=1079.238,127.608,430.460,174.230,23.178,153.979
C00872=1079.245,127.889,430.437,174.232,23.181,153.979
C00873=1079.250,128.138,430.418,174.234,23.183,153.979
C00874=1079.256,128.387,430.398,174.236,23.185,153.980
C00875=1079.262,128.637,430.379,174.238,23.187,153.980
C00876=1079.268,128.885,430.359,174.240,23.190,153.980
C00877=1079.274,129.135,430.340,174.241,23.192,153.980
C00878=1079.279,129.384,430.319,174.244,23.194,153.980
C00879=1079.285,129.633,430.299,174.245,23.196,153.981
C00880=1079.291,129.882,430.280,174.247,23.199,153.981
C00881=1079.297,130.131,430.260,174.249,23.201,153.981
C00882=1079.302,130.380,430.241,174.251,23.203,153.981
C00883=1079.308,130.630,430.220,174.253,23.206,153.981
C00884=1079.314,130.878,430.200,174.255,23.207,153.981
C00885=1079.319,131.128,430.181,174.257,23.210,153.982
C00886=1079.325,131.377,430.161,174.258,23.212,153.982
C00887=1079.330,131.626,430.140,174.261,23.214,153.982
C00888=1079.336,131.875,430.121,174.262,23.216,153.982
C00889=1079.342,132.124,430.101,174.264,23.218,153.982
C00890=1079.348,132.373,430.081,174.266,23.221,153.983
C00891=1079.353,132.623,430.061,174.268,23.223,153.983
C00892=1079.360,132.872,430.041,174.270,23.226,153.983
C00893=1079.365,133.121,430.020,174.272,23.228,153.983
C00894=1079.371,133.370,430.000,174.274,23.230,153.983
C00895=1079.376,133.620,429.981,174.275,23.232,153.984
C00896=1079.382,133.869,429.961,174.278,23.235,153.984
C00897=1079.388,134.117,429.941,174.279,23.236,153.984
C00898=1079.393,134.367,429.920,174.281,23.239,153.984
C00899=1079.399,134.616,429.901,174.284,23.242,153.984
C00900=1079.404,134.865,429.880,174.285,23.243,153.985
C00901=1079.410,135.114,429.860,174.287,23.246,153.985
C00902=1079.415,135.363,429.840,174.289,23.248,153.985
C00903=1079.421,135.612,429.820,174.291,23.250,153.985
C00904=1079.426,135.862,429.800,174.292,23.253,153.985
C00905=1079.432,136.110,429.780,174.295,23.255,153.986
C00906=1079.438,136.360,429.760,174.297,23.257,153.986
C00907=1079.444,136.608,429.740,174.298,23.260,153.986
C00908=1079.449,136.858,429.719,174.301,23.262,153.986
C00909=1079.455,137.107,429.699,174.302,23.264,153.986
C00910=1079.461,137.356,429.678,174.304,23.266,153.987
C00911=1079.466,137.606,429.659,174.306,23.268,153.987
C00912=1079.472,137.855,429.638,174.308,23.271,153.987
C00913=1079.478,138.103,429.618,174.310,23.273,153.987
C00914=1079.483,138.353,429.598,174.312,23.275,153.987
C00915=1079.489,138.601,429.578,174.314,23.277,153.987
C00916=1079.494,138.851,429.557,174.315,23.280,153.988
C00917=1079.501,139.100,429.537,174.318,23.282,153.988
C00918=1079.506,139.349,429.516,174.320,23.284,153.988
C00919=1079.512,139.598,429.496,174.321,23.286,153.988
C00920=1079.517,139.847,429.476,174.324,23.289,153.988
C00921=1079.523,140.096,429.456,174.325,23.291,153.989
C00922=1079.528,140.345,429.435,174.327,23.293,153.989
C00923=1079.534,140.594,429.415,174.330,23.296,153.989
C00924=1079.540,140.844,429.395,174.331,23.298,153.989
C00925=1079.546,141.093,429.374,174.333,23.300,153.989
C00926=1079.551,141.342,429.353,174.335,23.302,153.990
C00927=1079.557,141.591,429.333,174.337,23.305,153.990
C00928=1079.562,141.840,429.313,174.339,23.307,153.990
C00929=1079.567,142.089,429.292,174.341,23.309,153.990
C00930=1079.573,142.338,429.272,174.343,23.311,153.990
C00931=1079.579,142.588,429.251,174.345,23.313,153.990
C00932=1079.584,142.837,429.231,174.347,23.315,153.991
C00933=1079.591,143.117,429.207,174.349,23.318,153.991
C00934=1079.597,143.398,429.185,174.351,23.321,153.991
C00935=1079.604,143.678,429.161,174.354,23.323,153.991
C00936=1079.610,143.958,429.139,174.356,23.326,153.992
C00937=1079.616,144.208,429.118,174.357,23.328,153.992
C00938=1079.621,144.456,429.097,174.360,23.330,153.992
C00939=1079.626,144.706,429.076,174.362,23.332,153.992
C00940=1079.632,144.954,429.056,174.363,23.335,153.992
C00941=1079.638,145.204,429.035,174.366,23.337,153.992
C00942=1079.644,145.453,429.015,174.368,23.339,153.993
C00943=1079.649,145.702,428.994,174.369,23.341,153.993
C00944=1079.655,145.951,428.974,174.372,23.344,153.993
C00945=1079.660,146.200,428.953,174.373,23.346,153.993
C00946=1079.666,146.450,428.932,174.375,23.348,153.993
C00947=1079.671,146.699,428.912,174.378,23.350,153.993
C00948=1079.678,146.947,428.891,174.379,23.353,153.994
C00949=1079.684,147.197,428.870,174.381,23.355,153.994
C00950=1079.689,147.446,428.849,174.384,23.357,153.994
C00951=1079.694,147.695,428.829,174.385,23.359,153.994
C00952=1079.700,147.943,428.808,174.388,23.361,153.994
C00953=1079.706,148.193,428.787,174.390,23.364,153.995
C00954=1079.712,148.442,428.767,174.391,23.366,153.995
C00955=1079.717,148.691,428.745,174.394,23.368,153.995
C00956=1079.722,148.940,428.725,174.396,23.370,153.995
C00957=1079.728,149.190,428.704,174.397,23.373,153.995
C00958=1079.734,149.438,428.683,174.400,23.375,153.995
C00959=1079.739,149.687,428.662,174.401,23.377,153.996
C00960=1079.746,149.937,428.642,174.403,23.379,153.996
C00961=1079.751,150.185,428.621,174.406,23.382,153.996
C00962=1079.756,150.434,428.600,174.407,23.384,153.996
C00963=1079.762,150.683,428.579,174.409,23.386,153.996
C00964=1079.768,150.933,428.558,174.412,23.388,153.996
C00965=1079.773,151.182,428.537,174.413,23.390,153.997
C00966=1079.779,151.430,428.516,174.415,23.393,153.997
C00967=1079.785,151.680,428.495,174.418,23.395,153.997
C00968=1079.790,151.929,428.474,174.419,23.397,153.997
C00969=1079.795,152.178,428.453,174.422,23.399,153.997
C00970=1079.802,152.427,428.432,174.424,23.402,153.998
C00971=1079.807,152.676,428.411,174.425,23.404,153.998
C00972=1079.812,152.925,428.390,174.428,23.406,153.998
C00973=1079.818,153.174,428.369,174.430,23.408,153.998
C00974=1079.824,153.423,428.348,174.431,23.410,153.998
C00975=1079.829,153.672,428.327,174.434,23.413,153.999
C00976=1079.835,153.921,428.305,174.436,23.415,153.999
C00977=1079.840,154.170,428.285,174.438,23.417,153.999
C00978=1079.846,154.419,428.264,174.440,23.419,153.999
C00979=1079.852,154.669,428.243,174.442,23.422,153.999
C00980=1079.857,154.917,428.221,174.444,23.424,153.999
C00981=1079.863,155.166,428.201,174.446,23.426,154.000
C00982=1079.869,155.415,428.179,174.448,23.428,154.000
C00983=1079.874,155.664,428.158,174.451,23.430,154.000
C00984=1079.880,155.914,428.137,174.452,23.432,154.000
C00985=1079.886,156.162,428.116,174.454,23.435,154.000
C00986=1079.891,156.411,428.095,174.457,23.437,154.000
C00987=1079.896,156.661,428.073,174.458,23.439,154.001
C00988=1079.902,156.909,428.052,174.460,23.441,154.001
C00989=1079.907,157.159,428.031,174.463,23.444,154.001
C00990=1079.913,157.408,428.009,174.465,23.446,154.001
C00991=1079.919,157.656,427.988,174.466,23.448,154.001
C00992=1079.925,157.906,427.967,174.469,23.450,154.001
C00993=1079.930,158.155,427.946,174.471,23.453,154.002
C00994=1079.936,158.403,427.925,174.473,23.454,154.002
C00995=1079.941,158.653,427.903,174.475,23.457,154.002
C00996=1079.947,158.902,427.882,174.477,23.459,154.002
C00997=1079.953,159.182,427.858,174.480,23.462,154.002
C00998=1079.960,159.462,427.834,174.482,23.464,154.003
C00999=1079.966,159.743,427.810,174.484,23.467,154.003
C01000=1079.973,160.023,427.786,174.487,23.469,154.003
C01001=1079.978,160.272,427.765,174.489,23.472,154.003
C01002=1079.984,160.521,427.742,174.490,23.474,154.003
C01003=1079.989,160.770,427.721,174.493,23.476,154.003
C01004=1079.995,161.020,427.700,174.495,23.478,154.004
C01005=1080.001,161.268,427.679,174.497,23.480,154.004
C01006=1080.006,161.517,427.658,174.499,23.482,154.004
C01007=1080.012,161.766,427.635,174.501,23.485,154.004
C01008=1080.017,162.015,427.614,174.503,23.487,154.004
C01009=1080.023,162.264,427.592,174.506,23.489,154.004
C01010=1080.028,162.513,427.571,174.507,23.491,154.005
C01011=1080.033,162.762,427.550,174.509,23.494,154.005
C01012=1080.039,163.011,427.528,174.512,23.496,154.005
C01013=1080.044,163.260,427.506,174.514,23.498,154.005
C01014=1080.050,163.509,427.484,174.515,23.501,154.005
C01015=1080.055,163.758,427.463,174.518,23.503,154.006
C01016=1080.061,164.007,427.441,174.520,23.505,154.006
C01017=1080.066,164.256,427.420,174.523,23.507,154.006
C01018=1080.071,164.505,427.398,174.524,23.510,154.006
C01019=1080.077,164.754,427.376,174.526,23.512,154.006
C01020=1080.082,165.003,427.354,174.529,23.514,154.006
C01021=1080.088,165.252,427.333,174.531,23.516,154.007
C01022=1080.093,165.501,427.311,174.532,23.519,154.007
C01023=1080.099,165.750,427.289,174.535,23.521,154.007
C01024=1080.104,165.999,427.267,174.537,23.523,154.007
C01025=1080.110,166.248,427.246,174.539,23.526,154.007
C01026=1080.115,166.497,427.224,174.541,23.527,154.007
C01027=1080.121,166.746,427.202,174.543,23.530,154.008
C01028=1080.126,166.995,427.180,174.545,23.532,154.008
C01029=1080.132,167.244,427.158,174.548,23.535,154.008
C01030=1080.137,167.493,427.137,174.549,23.536,154.008
C01031=1080.143,167.742,427.115,174.551,23.539,154.008
C01032=1080.148,167.991,427.093,174.554,23.541,154.009
C01033=1080.154,168.240,427.071,174.556,23.544,154.009
C01034=1080.159,168.489,427.050,174.559,23.546,154.009
C01035=1080.165,168.738,427.027,174.560,23.548,154.009
C01036=1080.170,168.986,427.006,174.562,23.550,154.009
C01037=1080.176,169.236,426.983,174.565,23.553,154.009
C01038=1080.182,169.485,426.962,174.567,23.555,154.010
C01039=1080.187,169.734,426.940,174.568,23.557,154.010
C01040=1080.192,169.983,426.918,174.571,23.559,154.010
C01041=1080.198,170.232,426.896,174.573,23.561,154.010
C01042=1080.204,170.481,426.873,174.575,23.563,154.010
C01043=1080.209,170.729,426.852,174.578,23.566,154.010
C01044=1080.215,170.979,426.830,174.579,23.568,154.011
C01045=1080.221,171.228,426.808,174.582,23.570,154.011
C01046=1080.226,171.476,426.786,174.584,23.572,154.011
C01047=1080.231,171.726,426.763,174.586,23.575,154.011
C01048=1080.237,171.974,426.742,174.589,23.577,154.011
C01049=1080.242,172.224,426.720,174.590,23.579,154.011
C01050=1080.249,172.472,426.698,174.592,23.582,154.012
C01051=1080.254,172.721,426.676,174.595,23.584,154.012
C01052=1080.259,172.971,426.654,174.597,23.586,154.012
C01053=1080.265,173.219,426.631,174.599,23.588,154.012
C01054=1080.270,173.468,426.609,174.601,23.590,154.012
C01055=1080.276,173.717,426.588,174.603,23.592,154.012
C01056=1080.282,173.967,426.565,174.606,23.594,154.012
C01057=1080.287,174.215,426.543,174.608,23.597,154.013
C01058=1080.293,174.464,426.521,174.610,23.599,154.013
C01059=1080.299,174.713,426.498,174.613,23.602,154.013
C01060=1080.304,174.962,426.476,174.614,23.604,154.013
C01061=1080.310,175.241,426.452,174.617,23.606,154.013
C01062=1080.317,175.522,426.427,174.620,23.608,154.013
C01063=1080.323,175.802,426.402,174.622,23.611,154.014
C01064=1080.329,176.081,426.376,174.624,23.613,154.014
C01065=1080.336,176.331,426.355,174.627,23.616,154.014
C01066=1080.341,176.579,426.332,174.629,23.618,154.014
C01067=1080.346,176.828,426.310,174.631,23.620,154.014
C01068=1080.352,177.077,426.288,174.633,23.622,154.014
C01069=1080.358,177.326,426.265,174.635,23.624,154.015
C01070=1080.363,177.575,426.243,174.638,23.626,154.015
C01071=1080.369,177.824,426.221,174.640,23.629,154.015
C01072=1080.375,178.073,426.199,174.642,23.631,154.015
C01073=1080.380,178.322,426.176,174.645,23.633,154.015
C01074=1080.386,178.570,426.153,174.647,23.635,154.015
C01075=1080.392,178.820,426.132,174.649,23.637,154.015
C01076=1080.398,179.068,426.109,174.651,23.639,154.016
C01077=1080.403,179.318,426.087,174.653,23.642,154.016
C01078=1080.409,179.567,426.064,174.656,23.644,154.016
C01079=1080.414,179.815,426.042,174.658,23.646,154.016
C01080=1080.420,180.064,426.019,174.660,23.649,154.016
C01081=1080.426,180.313,425.996,174.663,23.651,154.016
C01082=1080.432,180.562,425.975,174.664,23.653,154.017
C01083=1080.438,180.811,425.952,174.667,23.655,154.017
C01084=1080.443,181.061,425.930,174.669,23.657,154.017
C01085=1080.448,181.309,425.907,174.671,23.659,154.017
C01086=1080.455,181.558,425.885,174.674,23.662,154.017
C01087=1080.460,181.807,425.862,174.676,23.664,154.017
C01088=1080.466,182.056,425.840,174.679,23.665,154.017
C01089=1080.472,182.305,425.817,174.681,23.668,154.017
C01090=1080.478,182.554,425.795,174.683,23.670,154.018
C01091=1080.483,182.803,425.772,174.685,23.672,154.018
C01092=1080.489,183.051,425.749,174.687,23.674,154.018
C01093=1080.494,183.300,425.726,174.690,23.676,154.018
C01094=1080.500,183.549,425.705,174.692,23.678,154.018
C01095=1080.506,183.798,425.682,174.694,23.681,154.018
C01096=1080.512,184.047,425.659,174.697,23.683,154.019
C01097=1080.518,184.296,425.636,174.699,23.685,154.019
C01098=1080.524,184.545,425.614,174.702,23.687,154.019
C01099=1080.530,184.794,425.591,174.704,23.690,154.019
C01100=1080.535,185.043,425.568,174.705,23.691,154.019
C01101=1080.540,185.291,425.546,174.708,23.694,154.019
C01102=1080.546,185.540,425.523,174.710,23.696,154.019
C01103=1080.551,185.789,425.499,174.712,23.699,154.020
C01104=1080.557,186.039,425.477,174.715,23.701,154.020
C01105=1080.562,186.288,425.454,174.717,23.703,154.020
C01106=1080.567,186.536,425.432,174.720,23.705,154.020
C01107=1080.573,186.785,425.409,174.722,23.707,154.020
C01108=1080.579,187.034,425.386,174.724,23.710,154.021
C01109=1080.584,187.283,425.362,174.726,23.712,154.021
C01110=1080.590,187.532,425.339,174.729,23.715,154.021
C01111=1080.595,187.781,425.316,174.730,23.716,154.021
C01112=1080.600,188.029,425.294,174.733,23.719,154.021
C01113=1080.606,188.278,425.271,174.735,23.721,154.021
C01114=1080.612,188.527,425.248,174.737,23.724,154.022
C01115=1080.617,188.776,425.224,174.740,23.726,154.022
C01116=1080.622,189.025,425.202,174.742,23.728,154.022
C01117=1080.628,189.274,425.179,174.744,23.730,154.022
C01118=1080.634,189.523,425.156,174.747,23.732,154.022
C01119=1080.640,189.771,425.133,174.749,23.735,154.022
C01120=1080.644,190.020,425.109,174.752,23.737,154.022
C01121=1080.650,190.269,425.086,174.754,23.740,154.023
C01122=1080.656,190.518,425.063,174.756,23.742,154.023
C01123=1080.661,190.767,425.040,174.759,23.744,154.023
C01124=1080.666,191.016,425.017,174.761,23.746,154.023
C01125=1080.673,191.295,424.991,174.763,23.748,154.023
C01126=1080.679,191.575,424.965,174.766,23.751,154.023
C01127=1080.685,191.855,424.939,174.769,23.754,154.024
C01128=1080.692,192.134,424.914,174.771,23.757,154.024
C01129=1080.697,192.383,424.891,174.773,23.759,154.024
C01130=1080.702,192.632,424.867,174.776,23.761,154.024
C01131=1080.708,192.881,424.843,174.778,23.763,154.024
C01132=1080.714,193.129,424.820,174.781,23.765,154.024
C01133=1080.720,193.378,424.797,174.783,23.768,154.025
C01134=1080.725,193.628,424.774,174.785,23.770,154.025
C01135=1080.731,193.877,424.751,174.788,23.772,154.025
C01136=1080.736,194.125,424.728,174.790,23.774,154.025
C01137=1080.742,194.374,424.704,174.793,23.776,154.025
C01138=1080.747,194.623,424.681,174.795,23.779,154.025
C01139=1080.753,194.872,424.658,174.797,23.781,154.026
C01140=1080.759,195.121,424.635,174.800,23.784,154.026
C01141=1080.764,195.369,424.611,174.802,23.786,154.026
C01142=1080.770,195.618,424.588,174.804,23.788,154.026
C01143=1080.775,195.867,424.565,174.807,23.790,154.026
C01144=1080.781,196.116,424.541,174.809,23.792,154.026
C01145=1080.787,196.365,424.518,174.811,23.795,154.026
C01146=1080.792,196.613,424.495,174.814,23.797,154.027
C01147=1080.797,196.863,424.471,174.816,23.799,154.027
C01148=1080.803,197.111,424.447,174.819,23.801,154.027
C01149=1080.809,197.360,424.425,174.821,23.803,154.027
C01150=1080.814,197.608,424.400,174.823,23.806,154.027
C01151=1080.820,197.857,424.377,174.826,23.808,154.027
C01152=1080.826,198.107,424.354,174.828,23.810,154.027
C01153=1080.832,198.355,424.330,174.831,23.812,154.028
C01154=1080.837,198.604,424.307,174.833,23.815,154.028
C01155=1080.843,198.853,424.284,174.835,23.817,154.028
C01156=1080.848,199.102,424.260,174.838,23.819,154.028
C01157=1080.854,199.351,424.237,174.840,23.822,154.028
C01158=1080.860,199.599,424.213,174.842,23.824,154.028
C01159=1080.865,199.848,424.189,174.845,23.826,154.029
C01160=1080.872,200.097,424.165,174.847,23.828,154.029
C01161=1080.878,200.346,424.142,174.850,23.830,154.029
C01162=1080.883,200.595,424.118,174.852,23.833,154.029
C01163=1080.889,200.844,424.095,174.854,23.835,154.029
C01164=1080.894,201.092,424.071,174.857,23.837,154.029
C01165=1080.900,201.341,424.048,174.859,23.839,154.029
C01166=1080.906,201.590,424.024,174.861,23.842,154.030
C01167=1080.911,201.839,424.001,174.864,23.844,154.030
C01168=1080.917,202.088,423.977,174.866,23.846,154.030
C01169=1080.922,202.337,423.953,174.869,23.848,154.030
C01170=1080.928,202.585,423.930,174.871,23.850,154.030
C01171=1080.934,202.834,423.905,174.873,23.853,154.030
C01172=1080.940,203.083,423.882,174.876,23.855,154.030
C01173=1080.945,203.332,423.858,174.878,23.857,154.031
C01174=1080.951,203.580,423.834,174.880,23.860,154.031
C01175=1080.956,203.829,423.811,174.883,23.862,154.031
C01176=1080.962,204.078,423.786,174.885,23.864,154.031
C01177=1080.967,204.327,423.763,174.889,23.867,154.031
C01178=1080.973,204.576,423.739,174.891,23.869,154.031
C01179=1080.979,204.825,423.715,174.893,23.871,154.032
C01180=1080.985,205.073,423.691,174.896,23.873,154.032
C01181=1080.990,205.322,423.667,174.898,23.876,154.032
C01182=1080.995,205.571,423.643,174.900,23.878,154.032
C01183=1081.001,205.819,423.619,174.903,23.880,154.032
C01184=1081.006,206.069,423.596,174.905,23.883,154.032
C01185=1081.012,206.318,423.571,174.907,23.885,154.033
C01186=1081.018,206.566,423.548,174.910,23.887,154.033
C01187=1081.023,206.814,423.523,174.912,23.889,154.033
C01188=1081.029,207.064,423.499,174.915,23.891,154.033
C01189=1081.052,208.096,423.400,175.012,23.943,154.031
C01190=1081.061,208.494,423.360,175.016,23.948,154.032
C01191=1081.071,208.891,423.321,175.019,23.954,154.032
C01192=1081.080,209.288,423.282,175.023,23.959,154.033
C01193=1081.089,209.686,423.243,175.027,23.964,154.034
C01194=1081.094,209.934,423.219,175.029,23.968,154.034
C01195=1081.100,210.183,423.193,175.032,23.971,154.034
C01196=1081.106,210.432,423.169,175.034,23.974,154.035
C01197=1081.111,210.681,423.144,175.036,23.977,154.035
C01198=1081.117,210.929,423.119,175.039,23.980,154.035
C01199=1081.123,211.178,423.095,175.041,23.984,154.036
C01200=1081.128,211.427,423.071,175.043,23.987,154.036
C01201=1081.134,211.676,423.045,175.045,23.990,154.037
C01202=1081.140,211.924,423.021,175.048,23.994,154.037
C01203=1081.145,212.174,422.996,175.050,23.996,154.037
C01204=1081.151,212.422,422.971,175.052,24.000,154.038
C01205=1081.156,212.671,422.946,175.055,24.003,154.038
C01206=1081.162,212.919,422.921,175.057,24.007,154.038
C01207=1081.168,213.168,422.897,175.060,24.010,154.039
C01208=1081.174,213.416,422.872,175.062,24.013,154.039
C01209=1081.179,213.666,422.847,175.065,24.017,154.040
C01210=1081.185,213.914,422.823,175.067,24.020,154.040
C01211=1081.190,214.163,422.797,175.069,24.023,154.040
C01212=1081.195,214.412,422.773,175.071,24.026,154.041
C01213=1081.202,214.660,422.747,175.074,24.029,154.041
C01214=1081.208,214.909,422.722,175.076,24.033,154.042
C01215=1081.213,215.158,422.698,175.078,24.036,154.042
C01216=1081.219,215.407,422.672,175.081,24.039,154.042
C01217=1081.224,215.655,422.647,175.083,24.043,154.043
C01218=1081.230,215.904,422.622,175.085,24.046,154.043
C01219=1081.235,216.152,422.598,175.087,24.049,154.044
C01220=1081.242,216.401,422.572,175.091,24.052,154.044
C01221=1081.247,216.649,422.547,175.093,24.055,154.044
C01222=1081.252,216.899,422.522,175.095,24.059,154.045
C01223=1081.259,217.147,422.497,175.098,24.062,154.045
C01224=1081.264,217.396,422.473,175.100,24.065,154.045
C01225=1081.269,217.645,422.447,175.102,24.069,154.046
C01226=1081.276,217.894,422.421,175.104,24.072,154.046
C01227=1081.281,218.142,422.397,175.107,24.075,154.046
C01228=1081.287,218.391,422.372,175.109,24.078,154.047
C01229=1081.292,218.639,422.346,175.111,24.081,154.047
C01230=1081.298,218.888,422.321,175.114,24.085,154.048
C01231=1081.304,219.137,422.296,175.116,24.088,154.048
C01232=1081.309,219.385,422.271,175.119,24.091,154.048
C01233=1081.315,219.634,422.245,175.121,24.094,154.049
C01234=1081.321,219.883,422.220,175.124,24.098,154.049
C01235=1081.327,220.131,422.196,175.126,24.101,154.050
C01236=1081.332,220.380,422.170,175.128,24.104,154.050
C01237=1081.338,220.629,422.145,175.131,24.108,154.050
C01238=1081.344,220.877,422.120,175.133,24.110,154.051
C01239=1081.349,221.126,422.094,175.135,24.114,154.051
C01240=1081.356,221.375,422.068,175.138,24.117,154.051
C01241=1081.362,221.624,422.044,175.140,24.121,154.052
C01242=1081.370,222.025,422.002,175.144,24.126,154.052
C01243=1081.380,222.426,421.961,175.148,24.131,154.053
C01244=1081.388,222.828,421.920,175.152,24.136,154.054
C01245=1081.398,223.229,421.879,175.155,24.141,154.054
C01246=1081.403,223.478,421.854,175.158,24.145,154.055
C01247=1081.409,223.727,421.828,175.161,24.148,154.055
C01248=1081.414,223.976,421.802,175.163,24.151,154.056
C01249=1081.420,224.224,421.778,175.166,24.155,154.056
C01250=1081.425,224.473,421.752,175.168,24.158,154.056
C01251=1081.432,224.721,421.726,175.170,24.161,154.057
C01252=1081.437,224.970,421.700,175.173,24.165,154.057
C01253=1081.442,225.219,421.675,175.175,24.168,154.057
C01254=1081.448,225.467,421.649,175.177,24.171,154.058
C01255=1081.454,225.716,421.623,175.180,24.175,154.058
C01256=1081.460,225.964,421.597,175.182,24.177,154.058
C01257=1081.465,226.213,421.572,175.185,24.181,154.059
C01258=1081.471,226.461,421.547,175.188,24.184,154.059
C01259=1081.477,226.710,421.521,175.190,24.187,154.060
C01260=1081.483,226.959,421.495,175.193,24.191,154.060
C01261=1081.488,227.208,421.469,175.195,24.194,154.060
C01262=1081.494,227.457,421.443,175.197,24.197,154.061
C01263=1081.500,227.704,421.418,175.200,24.200,154.061
C01264=1081.505,227.953,421.392,175.202,24.204,154.062
C01265=1081.511,228.202,421.366,175.204,24.207,154.062
C01266=1081.517,228.451,421.340,175.207,24.210,154.062
C01267=1081.522,228.700,421.315,175.209,24.214,154.063
C01268=1081.529,228.948,421.289,175.211,24.217,154.063
C01269=1081.534,229.196,421.263,175.215,24.220,154.063
C01270=1081.539,229.445,421.237,175.217,24.223,154.064
C01271=1081.545,229.694,421.212,175.220,24.227,154.064
C01272=1081.551,229.942,421.185,175.222,24.230,154.065
C01273=1081.557,230.191,421.160,175.224,24.233,154.065
C01274=1081.563,230.440,421.134,175.227,24.236,154.065
C01275=1081.569,230.688,421.107,175.229,24.239,154.066
C01276=1081.573,230.936,421.082,175.231,24.243,154.066
C01277=1081.580,231.185,421.056,175.234,24.246,154.066
C01278=1081.585,231.433,421.030,175.236,24.249,154.067
C01279=1081.591,231.682,421.004,175.239,24.253,154.067
C01280=1081.596,231.931,420.978,175.242,24.256,154.068
C01281=1081.602,232.180,420.951,175.244,24.259,154.068
C01282=1081.608,232.429,420.925,175.247,24.263,154.068
C01283=1081.614,232.677,420.899,175.249,24.266,154.069
C01284=1081.620,232.926,420.873,175.251,24.269,154.069
C01285=1081.624,233.174,420.848,175.254,24.272,154.069
C01286=1081.630,233.422,420.821,175.256,24.276,154.070
C01287=1081.636,233.671,420.795,175.259,24.279,154.070
C01288=1081.641,233.920,420.768,175.261,24.282,154.071
C01289=1081.648,234.168,420.743,175.263,24.286,154.071
C01290=1081.653,234.417,420.716,175.266,24.289,154.071
C01291=1081.659,234.666,420.690,175.268,24.292,154.072
C01292=1081.665,234.914,420.664,175.272,24.295,154.072
C01293=1081.670,235.163,420.638,175.274,24.299,154.073
C01294=1081.679,235.556,420.596,175.277,24.304,154.073
C01295=1081.687,235.949,420.554,175.282,24.309,154.074
C01296=1081.697,236.342,420.513,175.285,24.314,154.074
C01297=1081.706,236.735,420.471,175.290,24.320,154.075
C01298=1081.712,236.983,420.445,175.292,24.323,154.075
C01299=1081.717,237.231,420.418,175.294,24.326,154.076
C01300=1081.723,237.480,420.392,175.297,24.330,154.076
C01301=1081.729,237.729,420.365,175.299,24.333,154.077
C01302=1081.734,237.977,420.339,175.302,24.336,154.077
C01303=1081.740,238.226,420.313,175.305,24.339,154.077
C01304=1081.746,238.474,420.286,175.308,24.343,154.078
C01305=1081.751,238.723,420.259,175.310,24.346,154.078
C01306=1081.757,238.971,420.233,175.312,24.349,154.079
C01307=1081.763,239.220,420.207,175.315,24.353,154.079
C01308=1081.768,239.468,420.180,175.317,24.356,154.079
C01309=1081.774,239.717,420.154,175.320,24.359,154.080
C01310=1081.780,239.965,420.127,175.322,24.362,154.080
C01311=1081.786,240.215,420.101,175.325,24.366,154.080
C01312=1081.792,240.463,420.074,175.327,24.369,154.081
C01313=1081.798,240.712,420.047,175.330,24.372,154.081
C01314=1081.803,240.960,420.021,175.333,24.376,154.082
C01315=1081.809,241.208,419.994,175.335,24.379,154.082
C01316=1081.814,241.457,419.967,175.338,24.382,154.082
C01317=1081.820,241.705,419.940,175.340,24.386,154.083
C01318=1081.826,241.954,419.914,175.343,24.389,154.083
C01319=1081.831,242.203,419.888,175.345,24.392,154.083
C01320=1081.837,242.451,419.861,175.348,24.395,154.084
C01321=1081.843,242.700,419.834,175.350,24.399,154.084
C01322=1081.849,242.948,419.807,175.353,24.402,154.085
C01323=1081.855,243.197,419.781,175.355,24.405,154.085
C01324=1081.860,243.446,419.753,175.358,24.408,154.085
C01325=1081.866,243.694,419.727,175.361,24.412,154.086
C01326=1081.871,243.942,419.700,175.363,24.415,154.086
C01327=1081.876,244.191,419.673,175.366,24.419,154.087
C01328=1081.882,244.439,419.646,175.368,24.422,154.087
C01329=1081.888,244.688,419.620,175.371,24.426,154.087
C01330=1081.894,244.937,419.593,175.373,24.429,154.088
C01331=1081.900,245.185,419.565,175.376,24.432,154.088
C01332=1081.905,245.433,419.538,175.378,24.435,154.089
C01333=1081.911,245.681,419.511,175.381,24.439,154.089
C01334=1081.916,245.930,419.484,175.383,24.442,154.089
C01335=1081.922,246.178,419.457,175.386,24.445,154.090
C01336=1081.928,246.427,419.431,175.389,24.448,154.090
C01337=1081.933,246.676,419.403,175.392,24.452,154.091
C01338=1081.939,246.925,419.376,175.394,24.455,154.091
C01339=1081.945,247.172,419.349,175.397,24.459,154.091
C01340=1081.950,247.421,419.322,175.399,24.462,154.092
C01341=1081.956,247.669,419.295,175.402,24.465,154.092
C01342=1081.961,247.918,419.268,175.404,24.469,154.093
C01343=1081.968,248.166,419.240,175.407,24.472,154.093
C01344=1081.973,248.415,419.213,175.409,24.475,154.093
C01345=1081.979,248.663,419.186,175.411,24.479,154.094
C01346=1081.987,249.050,419.143,175.416,24.484,154.094
C01347=1081.995,249.436,419.102,175.419,24.489,154.095
C01348=1082.005,249.822,419.059,175.424,24.495,154.096
C01349=1082.013,250.208,419.017,175.428,24.500,154.096
C01350=1082.019,250.457,418.989,175.431,24.503,154.097
C01351=1082.025,250.705,418.962,175.433,24.506,154.097
C01352=1082.030,250.954,418.934,175.436,24.510,154.097
C01353=1082.036,251.202,418.908,175.438,24.513,154.098
C01354=1082.042,251.451,418.880,175.441,24.517,154.098
C01355=1082.047,251.699,418.853,175.443,24.520,154.099
C01356=1082.053,251.947,418.825,175.446,24.523,154.099
C01357=1082.058,252.196,418.798,175.448,24.527,154.099
C01358=1082.064,252.444,418.770,175.451,24.530,154.100
C01359=1082.070,252.693,418.743,175.454,24.533,154.100
C01360=1082.075,252.941,418.716,175.457,24.537,154.101
C01361=1082.081,253.189,418.688,175.459,24.540,154.101
C01362=1082.087,253.438,418.660,175.462,24.544,154.102
C01363=1082.092,253.686,418.633,175.464,24.547,154.102
C01364=1082.098,253.934,418.605,175.467,24.550,154.102
C01365=1082.104,254.183,418.578,175.470,24.554,154.103
C01366=1082.109,254.432,418.550,175.472,24.557,154.103
C01367=1082.114,254.680,418.523,175.475,24.560,154.103
C01368=1082.121,254.929,418.495,175.477,24.564,154.104
C01369=1082.126,255.177,418.467,175.480,24.567,154.104
C01370=1082.132,255.425,418.440,175.482,24.570,154.105
C01371=1082.138,255.674,418.412,175.486,24.574,154.105
C01372=1082.144,255.922,418.384,175.488,24.577,154.105
C01373=1082.149,256.171,418.357,175.491,24.581,154.106
C01374=1082.155,256.419,418.329,175.493,24.584,154.106
C01375=1082.161,256.667,418.301,175.496,24.587,154.107
C01376=1082.166,256.916,418.274,175.498,24.590,154.107
C01377=1082.172,257.164,418.246,175.501,24.594,154.107
C01378=1082.178,257.413,418.218,175.504,24.598,154.108
C01379=1082.184,257.661,418.190,175.506,24.601,154.108
C01380=1082.189,257.909,418.163,175.509,24.604,154.109
C01381=1082.195,258.158,418.135,175.511,24.607,154.109
C01382=1082.201,258.406,418.107,175.515,24.611,154.109
C01383=1082.207,258.655,418.079,175.517,24.614,154.110
C01384=1082.213,258.903,418.051,175.520,24.618,154.110
C01385=1082.218,259.152,418.024,175.523,24.621,154.111
C01386=1082.224,259.400,417.997,175.525,24.624,154.111
C01387=1082.230,259.648,417.968,175.528,24.628,154.111
C01388=1082.236,259.896,417.940,175.530,24.631,154.112
C01389=1082.242,260.145,417.912,175.533,24.635,154.112
C01390=1082.248,260.393,417.885,175.535,24.638,154.113
C01391=1082.254,260.642,417.856,175.538,24.641,154.113
C01392=1082.259,260.890,417.828,175.541,24.645,154.113
C01393=1082.265,261.139,417.800,175.544,24.648,154.114
C01394=1082.271,261.386,417.773,175.547,24.652,154.114
C01395=1082.277,261.635,417.744,175.549,24.655,154.115
C01396=1082.282,261.883,417.716,175.552,24.658,154.115
C01397=1082.288,262.132,417.688,175.554,24.661,154.115
C01398=1082.297,262.515,417.645,175.559,24.666,154.116
C01399=1082.306,262.899,417.602,175.563,24.672,154.117
C01400=1082.315,263.282,417.559,175.567,24.677,154.117
C01401=1082.325,263.666,417.515,175.571,24.682,154.118
C01402=1082.330,263.914,417.488,175.574,24.685,154.118
C01403=1082.336,264.162,417.458,175.577,24.689,154.119
C01404=1082.342,264.410,417.431,175.579,24.692,154.119
C01405=1082.348,264.659,417.402,175.582,24.696,154.119
C01406=1082.353,264.907,417.374,175.585,24.699,154.120
C01407=1082.359,265.156,417.346,175.587,24.702,154.120
C01408=1082.364,265.404,417.318,175.590,24.706,154.121
C01409=1082.370,265.652,417.289,175.592,24.709,154.121
C01410=1082.376,265.901,417.261,175.595,24.712,154.121
C01411=1082.382,266.149,417.233,175.598,24.716,154.122
C01412=1082.388,266.397,417.204,175.600,24.720,154.122
C01413=1082.393,266.645,417.176,175.603,24.723,154.123
C01414=1082.399,266.894,417.147,175.606,24.726,154.123
C01415=1082.405,267.143,417.118,175.609,24.730,154.124
C01416=1082.410,267.391,417.090,175.612,24.733,154.124
C01417=1082.416,267.639,417.061,175.614,24.736,154.124
C01418=1082.421,267.887,417.033,175.617,24.740,154.125
C01419=1082.427,268.136,417.005,175.620,24.744,154.125
C01420=1082.434,268.384,416.976,175.622,24.747,154.126
C01421=1082.439,268.632,416.948,175.625,24.751,154.126
C01422=1082.445,268.880,416.919,175.627,24.754,154.127
C01423=1082.451,269.129,416.891,175.630,24.757,154.127
C01424=1082.456,269.377,416.862,175.633,24.761,154.127
C01425=1082.462,269.625,416.833,175.636,24.764,154.128
C01426=1082.467,269.873,416.805,175.639,24.768,154.128
C01427=1082.474,270.121,416.776,175.642,24.771,154.128
C01428=1082.480,270.370,416.748,175.644,24.775,154.129
C01429=1082.484,270.618,416.719,175.647,24.778,154.129
C01430=1082.490,270.867,416.690,175.650,24.782,154.130
C01431=1082.497,271.115,416.661,175.652,24.785,154.130
C01432=1082.502,271.363,416.633,175.655,24.788,154.131
C01433=1082.508,271.611,416.604,175.658,24.792,154.131
C01434=1082.513,271.860,416.575,175.660,24.796,154.132
C01435=1082.520,272.108,416.546,175.663,24.799,154.132
C01436=1082.525,272.356,416.518,175.665,24.802,154.132
C01437=1082.531,272.605,416.489,175.669,24.806,154.133
C01438=1082.537,272.853,416.460,175.672,24.809,154.133
C01439=1082.542,273.101,416.432,175.674,24.812,154.134
C01440=1082.548,273.349,416.403,175.677,24.816,154.134
C01441=1082.554,273.597,416.373,175.680,24.820,154.135
C01442=1082.560,273.846,416.345,175.682,24.823,154.135
C01443=1082.565,274.094,416.316,175.685,24.827,154.135
C01444=1082.571,274.342,416.286,175.688,24.830,154.136
C01445=1082.577,274.591,416.258,175.690,24.834,154.136
C01446=1082.582,274.839,416.229,175.693,24.837,154.137
C01447=1082.588,275.087,416.200,175.696,24.841,154.137
C01448=1082.594,275.335,416.171,175.698,24.844,154.137
C01449=1082.600,275.584,416.142,175.701,24.848,154.138
C01450=1082.609,275.970,416.096,175.706,24.853,154.139
C01451=1082.618,276.356,416.051,175.710,24.859,154.139
C01452=1082.626,276.743,416.006,175.714,24.864,154.140
C01453=1082.636,277.129,415.961,175.719,24.870,154.141
C01454=1082.641,277.377,415.931,175.722,24.873,154.141
C01455=1082.647,277.625,415.902,175.724,24.877,154.142
C01456=1082.652,277.874,415.873,175.727,24.880,154.142
C01457=1082.659,278.122,415.844,175.730,24.884,154.142
C01458=1082.664,278.370,415.814,175.733,24.887,154.143
C01459=1082.670,278.618,415.785,175.735,24.891,154.143
C01460=1082.675,278.866,415.756,175.738,24.894,154.144
C01461=1082.682,279.114,415.727,175.741,24.898,154.144
C01462=1082.687,279.363,415.697,175.743,24.902,154.145
C01463=1082.693,279.611,415.668,175.746,24.905,154.145
C01464=1082.699,279.859,415.638,175.749,24.909,154.145
C01465=1082.705,280.107,415.609,175.752,24.912,154.146
C01466=1082.710,280.355,415.580,175.755,24.916,154.146
C01467=1082.715,280.603,415.550,175.758,24.919,154.147
C01468=1082.722,280.852,415.521,175.761,24.923,154.147
C01469=1082.727,281.100,415.492,175.763,24.926,154.148
C01470=1082.733,281.348,415.463,175.766,24.930,154.148
C01471=1082.739,281.597,415.433,175.769,24.933,154.148
C01472=1082.745,281.845,415.403,175.771,24.937,154.149
C01473=1082.750,282.093,415.374,175.774,24.940,154.149
C01474=1082.756,282.340,415.344,175.777,24.944,154.150
C01475=1082.761,282.589,415.315,175.780,24.948,154.150
C01476=1082.767,282.837,415.285,175.782,24.951,154.151
C01477=1082.773,283.086,415.255,175.785,24.955,154.151
C01478=1082.779,283.334,415.226,175.788,24.959,154.152
C01479=1082.785,283.582,415.196,175.791,24.963,154.152
C01480=1082.790,283.830,415.166,175.793,24.966,154.153
C01481=1082.796,284.078,415.137,175.796,24.969,154.153
C01482=1082.802,284.326,415.107,175.799,24.973,154.154
C01483=1082.808,284.574,415.077,175.803,24.977,154.154
C01484=1082.813,284.823,415.048,175.805,24.980,154.155
C01485=1082.819,285.071,415.018,175.808,24.984,154.155
C01486=1082.825,285.318,414.989,175.811,24.988,154.155
C01487=1082.830,285.567,414.959,175.814,24.991,154.156
C01488=1082.836,285.814,414.929,175.816,24.994,154.156
C01489=1082.841,286.063,414.899,175.819,24.998,154.157
C01490=1082.847,286.311,414.869,175.822,25.002,154.157
C01491=1082.854,286.559,414.840,175.825,25.006,154.158
C01492=1082.859,286.807,414.810,175.827,25.009,154.158
C01493=1082.865,287.055,414.780,175.830,25.012,154.159
C01494=1082.870,287.303,414.750,175.833,25.016,154.159
C01495=1082.876,287.551,414.720,175.836,25.020,154.159
C01496=1082.882,287.800,414.690,175.838,25.024,154.160
C01497=1082.889,288.048,414.660,175.841,25.027,154.160
C01498=1082.894,288.296,414.630,175.844,25.031,154.161
C01499=1082.900,288.544,414.600,175.847,25.035,154.161
C01500=1082.906,288.793,414.570,175.850,25.038,154.162
C01501=1082.912,289.040,414.540,175.853,25.042,154.162
C01502=1082.921,289.437,414.493,175.857,25.047,154.163
C01503=1082.930,289.833,414.445,175.862,25.053,154.164
C01504=1082.939,290.228,414.396,175.866,25.059,154.164
C01505=1082.948,290.625,414.349,175.871,25.065,154.165
C01506=1082.954,290.873,414.318,175.874,25.069,154.166
C01507=1082.960,291.121,414.288,175.877,25.073,154.166
C01508=1082.965,291.369,414.258,175.880,25.076,154.167
C01509=1082.971,291.617,414.228,175.883,25.080,154.167
C01510=1082.977,291.865,414.198,175.885,25.084,154.168
C01511=1082.983,292.113,414.167,175.888,25.087,154.168
C01512=1082.989,292.362,414.137,175.891,25.091,154.169
C01513=1082.995,292.610,414.107,175.894,25.095,154.169
C01514=1083.001,292.857,414.077,175.897,25.099,154.170
C01515=1083.006,293.105,414.046,175.899,25.102,154.170
C01516=1083.012,293.353,414.015,175.902,25.106,154.170
C01517=1083.017,293.602,413.986,175.905,25.110,154.171
C01518=1083.023,293.850,413.955,175.908,25.113,154.171
C01519=1083.029,294.097,413.925,175.911,25.117,154.172
C01520=1083.035,294.346,413.894,175.913,25.120,154.172
C01521=1083.041,294.594,413.864,175.916,25.124,154.173
C01522=1083.047,294.842,413.833,175.919,25.128,154.173
C01523=1083.053,295.089,413.803,175.922,25.132,154.174
C01524=1083.058,295.337,413.772,175.925,25.136,154.174
C01525=1083.064,295.586,413.741,175.928,25.140,154.175
C01526=1083.070,295.834,413.711,175.930,25.143,154.175
C01527=1083.076,296.082,413.681,175.933,25.147,154.176
C01528=1083.081,296.329,413.650,175.936,25.151,154.176
C01529=1083.087,296.578,413.619,175.939,25.154,154.177
C01530=1083.092,296.825,413.589,175.942,25.158,154.177
C01531=1083.099,297.074,413.558,175.945,25.162,154.178
C01532=1083.105,297.322,413.528,175.949,25.165,154.178
C01533=1083.110,297.570,413.497,175.951,25.169,154.179
C01534=1083.116,297.818,413.467,175.954,25.173,154.179
C01535=1083.122,298.066,413.436,175.957,25.177,154.180
C01536=1083.127,298.314,413.405,175.960,25.180,154.180
C01537=1083.133,298.562,413.375,175.963,25.184,154.181
C01538=1083.138,298.810,413.343,175.966,25.188,154.181
C01539=1083.144,299.058,413.313,175.968,25.192,154.182
C01540=1083.150,299.306,413.281,175.971,25.196,154.182
C01541=1083.156,299.554,413.251,175.974,25.200,154.183
C01542=1083.161,299.802,413.220,175.977,25.204,154.183
C01543=1083.167,300.050,413.189,175.980,25.208,154.184
C01544=1083.172,300.298,413.158,175.983,25.212,154.184
C01545=1083.178,300.546,413.127,175.986,25.215,154.185
C01546=1083.184,300.794,413.096,175.989,25.219,154.185
C01547=1083.189,301.042,413.065,175.991,25.223,154.186
C01548=1083.195,301.290,413.034,175.994,25.227,154.186
C01549=1083.201,301.538,413.004,175.997,25.231,154.187
C01550=1083.206,301.786,412.972,176.000,25.235,154.187
C01551=1083.212,302.033,412.942,176.003,25.239,154.188
C01552=1083.218,302.281,412.910,176.006,25.243,154.189
C01553=1083.224,302.530,412.879,176.009,25.247,154.189
C01554=1083.233,302.940,412.828,176.013,25.253,154.190
C01555=1083.243,303.350,412.776,176.018,25.259,154.191
C01556=1083.252,303.760,412.725,176.023,25.266,154.192
C01557=1083.261,304.171,412.673,176.028,25.273,154.193
C01558=1083.267,304.418,412.642,176.030,25.276,154.193
C01559=1083.273,304.667,412.611,176.033,25.280,154.194
C01560=1083.279,304.914,412.579,176.036,25.284,154.194
C01561=1083.284,305.162,412.549,176.039,25.288,154.195
C01562=1083.290,305.410,412.517,176.042,25.291,154.195
C01563=1083.296,305.657,412.486,176.045,25.295,154.196
C01564=1083.302,305.906,412.455,176.048,25.299,154.196
C01565=1083.308,306.154,412.423,176.051,25.303,154.197
C01566=1083.313,306.402,412.393,176.054,25.307,154.197
C01567=1083.319,306.650,412.361,176.057,25.311,154.198
C01568=1083.325,306.897,412.330,176.060,25.315,154.198
C01569=1083.331,307.146,412.298,176.063,25.319,154.199
C01570=1083.337,307.393,412.267,176.066,25.323,154.199
C01571=1083.343,307.641,412.235,176.069,25.327,154.200
C01572=1083.349,307.889,412.203,176.071,25.331,154.200
C01573=1083.354,308.138,412.172,176.074,25.335,154.201
C01574=1083.360,308.385,412.141,176.077,25.338,154.202
C01575=1083.366,308.633,412.109,176.080,25.342,154.202
C01576=1083.372,308.881,412.077,176.083,25.346,154.203
C01577=1083.378,309.129,412.047,176.086,25.350,154.203
C01578=1083.384,309.377,412.015,176.089,25.354,154.204
C01579=1083.390,309.625,411.983,176.092,25.358,154.204
C01580=1083.395,309.872,411.951,176.095,25.362,154.205
C01581=1083.402,310.120,411.920,176.098,25.367,154.205
C01582=1083.407,310.368,411.888,176.101,25.371,154.206
C01583=1083.413,310.617,411.857,176.104,25.374,154.206
C01584=1083.419,310.864,411.826,176.107,25.378,154.207
C01585=1083.425,311.112,411.794,176.110,25.382,154.207
C01586=1083.431,311.360,411.762,176.113,25.386,154.208
C01587=1083.436,311.608,411.730,176.116,25.390,154.209
C01588=1083.443,311.856,411.699,176.119,25.394,154.209
C01589=1083.448,312.103,411.667,176.122,25.398,154.210
C01590=1083.454,312.351,411.635,176.125,25.402,154.210
C01591=1083.460,312.600,411.603,176.128,25.406,154.211
C01592=1083.466,312.847,411.572,176.131,25.410,154.211
C01593=1083.472,313.095,411.540,176.134,25.414,154.212
C01594=1083.478,313.343,411.508,176.137,25.418,154.212
C01595=1083.484,313.591,411.476,176.140,25.422,154.213
C01596=1083.491,313.839,411.445,176.143,25.426,154.213
C01597=1083.497,314.087,411.413,176.146,25.430,154.214
C01598=1083.502,314.334,411.381,176.149,25.434,154.215
C01599=1083.508,314.583,411.349,176.152,25.438,154.215
C01600=1083.514,314.830,411.316,176.154,25.442,154.216
C01601=1083.520,315.078,411.284,176.157,25.446,154.216
C01602=1083.526,315.326,411.253,176.160,25.450,154.217
C01603=1083.532,315.574,411.221,176.163,25.454,154.217
C01604=1083.537,315.822,411.189,176.166,25.458,154.218
C01605=1083.543,316.069,411.156,176.169,25.463,154.219
C01606=1083.552,316.482,411.102,176.174,25.470,154.220
C01607=1083.562,316.896,411.049,176.179,25.477,154.221
C01608=1083.571,317.309,410.995,176.184,25.483,154.222
C01609=1083.581,317.722,410.941,176.189,25.490,154.223
C01610=1083.587,317.971,410.909,176.192,25.495,154.223
C01611=1083.592,318.218,410.876,176.195,25.499,154.224
C01612=1083.598,318.466,410.844,176.198,25.503,154.224
C01613=1083.604,318.714,410.812,176.201,25.507,154.225
C01614=1083.609,318.961,410.780,176.204,25.511,154.226
C01615=1083.615,319.210,410.747,176.207,25.516,154.226
C01616=1083.621,319.457,410.714,176.210,25.520,154.227
C01617=1083.626,319.705,410.683,176.212,25.524,154.227
C01618=1083.632,319.953,410.651,176.215,25.528,154.228
C01619=1083.638,320.201,410.617,176.218,25.532,154.229
C01620=1083.644,320.449,410.585,176.221,25.536,154.229
C01621=1083.650,320.696,410.553,176.224,25.541,154.230
C01622=1083.656,320.944,410.521,176.227,25.545,154.231
C01623=1083.661,321.192,410.488,176.231,25.550,154.231
C01624=1083.667,321.440,410.455,176.234,25.554,154.232
C01625=1083.673,321.688,410.423,176.237,25.558,154.232
C01626=1083.678,321.935,410.390,176.240,25.562,154.233
C01627=1083.684,322.183,410.358,176.243,25.567,154.234
C01628=1083.691,322.431,410.325,176.246,25.571,154.234
C01629=1083.696,322.679,410.292,176.249,25.575,154.235
C01630=1083.702,322.927,410.260,176.252,25.579,154.235
C01631=1083.709,323.175,410.227,176.255,25.583,154.236
C01632=1083.713,323.422,410.194,176.258,25.588,154.237
C01633=1083.719,323.670,410.162,176.261,25.592,154.237
C01634=1083.726,323.918,410.129,176.264,25.596,154.238
C01635=1083.731,324.165,410.096,176.266,25.600,154.238
C01636=1083.737,324.414,410.064,176.269,25.605,154.239
C01637=1083.743,324.662,410.031,176.272,25.609,154.240
C01638=1083.749,324.909,409.998,176.276,25.614,154.240
C01639=1083.755,325.157,409.965,176.279,25.618,154.241
C01640=1083.761,325.405,409.932,176.282,25.622,154.242
C01641=1083.767,325.653,409.900,176.285,25.626,154.242
C01642=1083.773,325.900,409.867,176.288,25.631,154.243
C01643=1083.778,326.148,409.834,176.291,25.635,154.244
C01644=1083.785,326.395,409.801,176.294,25.639,154.244
C01645=1083.790,326.643,409.768,176.297,25.644,154.245
C01646=1083.796,326.891,409.735,176.300,25.648,154.245
C01647=1083.802,327.139,409.702,176.303,25.652,154.246
C01648=1083.808,327.386,409.669,176.306,25.657,154.247
C01649=1083.815,327.634,409.636,176.309,25.661,154.247
C01650=1083.820,327.882,409.603,176.312,25.665,154.248
C01651=1083.826,328.129,409.570,176.315,25.670,154.249
C01652=1083.832,328.377,409.537,176.318,25.674,154.249
C01653=1083.838,328.625,409.504,176.321,25.678,154.250
C01654=1083.844,328.873,409.471,176.324,25.683,154.251
C01655=1083.851,329.121,409.438,176.327,25.687,154.251
C01656=1083.856,329.369,409.404,176.331,25.691,154.252
C01657=1083.862,329.617,409.372,176.334,25.696,154.252
C01658=1083.872,330.023,409.317,176.338,25.703,154.254
C01659=1083.882,330.429,409.263,176.343,25.710,154.255
C01660=1083.892,330.835,409.209,176.349,25.717,154.256
C01661=1083.902,331.243,409.153,176.354,25.725,154.257
C01662=1083.908,331.490,409.121,176.357,25.729,154.257
C01663=1083.914,331.738,409.087,176.360,25.733,154.258
C01664=1083.919,331.986,409.054,176.363,25.738,154.259
C01665=1083.926,332.234,409.021,176.366,25.743,154.259
C01666=1083.932,332.481,408.987,176.369,25.747,154.260
C01667=1083.937,332.729,408.954,176.372,25.752,154.261
C01668=1083.943,332.977,408.921,176.375,25.756,154.261
C01669=1083.949,333.224,408.887,176.378,25.761,154.262
C01670=1083.955,333.472,408.854,176.381,25.765,154.263
C01671=1083.961,333.720,408.820,176.385,25.770,154.264
C01672=1083.967,333.967,408.786,176.388,25.775,154.264
C01673=1083.972,334.215,408.753,176.390,25.779,154.265
C01674=1083.978,334.463,408.719,176.393,25.783,154.266
C01675=1083.984,334.711,408.685,176.396,25.788,154.266
C01676=1083.990,334.957,408.652,176.399,25.793,154.267
C01677=1083.996,335.205,408.619,176.403,25.797,154.268
C01678=1084.002,335.454,408.585,176.406,25.802,154.268
C01679=1084.008,335.701,408.551,176.409,25.807,154.269
C01680=1084.014,335.949,408.517,176.412,25.811,154.270
C01681=1084.019,336.196,408.483,176.416,25.816,154.270
C01682=1084.025,336.444,408.449,176.418,25.821,154.271
C01683=1084.032,336.691,408.417,176.421,25.825,154.272
C01684=1084.038,336.939,408.382,176.424,25.830,154.273
C01685=1084.044,337.187,408.349,176.427,25.834,154.273
C01686=1084.049,337.435,408.315,176.431,25.839,154.274
C01687=1084.055,337.682,408.281,176.434,25.844,154.275
C01688=1084.061,337.930,408.247,176.437,25.848,154.275
C01689=1084.067,338.178,408.213,176.440,25.852,154.276
C01690=1084.073,338.425,408.179,176.443,25.858,154.277
C01691=1084.079,338.673,408.146,176.446,25.863,154.278
C01692=1084.085,338.921,408.111,176.449,25.867,154.278
C01693=1084.091,339.168,408.077,176.452,25.872,154.279
C01694=1084.097,339.416,408.044,176.456,25.876,154.280
C01695=1084.102,339.663,408.010,176.459,25.881,154.281
C01696=1084.109,339.911,407.975,176.461,25.886,154.281
C01697=1084.115,340.159,407.941,176.464,25.891,154.282
C01698=1084.120,340.406,407.907,176.468,25.896,154.283
C01699=1084.126,340.653,407.873,176.471,25.900,154.284
C01700=1084.132,340.902,407.839,176.474,25.905,154.284
C01701=1084.138,341.149,407.805,176.477,25.910,154.285
C01702=1084.144,341.397,407.771,176.480,25.915,154.286
C01703=1084.150,341.645,407.736,176.483,25.919,154.287
C01704=1084.156,341.892,407.702,176.486,25.924,154.287
C01705=1084.162,342.139,407.668,176.489,25.929,154.288
C01706=1084.168,342.388,407.633,176.493,25.934,154.289
C01707=1084.173,342.635,407.599,176.496,25.939,154.290
C01708=1084.179,342.882,407.565,176.499,25.944,154.290
C01709=1084.186,343.130,407.531,176.502,25.949,154.291
C01710=1084.195,343.531,407.476,176.507,25.957,154.292
C01711=1084.205,343.932,407.420,176.512,25.964,154.294
C01712=1084.215,344.332,407.364,176.517,25.972,154.295
C01713=1084.224,344.733,407.308,176.522,25.980,154.296
C01714=1084.230,344.981,407.274,176.526,25.985,154.297
C01715=1084.236,345.229,407.239,176.528,25.990,154.298
C01716=1084.242,345.476,407.205,176.531,25.995,154.298
C01717=1084.248,345.723,407.170,176.535,26.000,154.299
C01718=1084.254,345.971,407.135,176.538,26.005,154.300
C01719=1084.260,346.219,407.101,176.541,26.010,154.301
C01720=1084.266,346.467,407.067,176.544,26.015,154.302
C01721=1084.272,346.714,407.031,176.547,26.020,154.302
C01722=1084.278,346.962,406.997,176.550,26.024,154.303
C01723=1084.283,347.209,406.962,176.554,26.030,154.304
C01724=1084.289,347.456,406.928,176.557,26.034,154.305
C01725=1084.296,347.704,406.893,176.560,26.039,154.306
C01726=1084.301,347.951,406.858,176.563,26.045,154.306
C01727=1084.308,348.199,406.823,176.566,26.050,154.307
C01728=1084.313,348.446,406.789,176.569,26.055,154.308
C01729=1084.319,348.694,406.754,176.573,26.060,154.309
C01730=1084.325,348.941,406.719,176.576,26.065,154.310
C01731=1084.331,349.189,406.685,176.579,26.070,154.311
C01732=1084.337,349.436,406.650,176.582,26.075,154.311
C01733=1084.343,349.684,406.615,176.585,26.080,154.312
C01734=1084.349,349.931,406.580,176.589,26.085,154.313
C01735=1084.355,350.179,406.545,176.591,26.090,154.314
C01736=1084.361,350.426,406.510,176.594,26.095,154.315
C01737=1084.367,350.674,406.475,176.598,26.100,154.315
C01738=1084.374,350.921,406.440,176.601,26.106,154.316
C01739=1084.379,351.168,406.405,176.605,26.111,154.317
C01740=1084.385,351.417,406.370,176.607,26.116,154.318
C01741=1084.391,351.663,406.335,176.610,26.121,154.319
C01742=1084.397,351.912,406.300,176.614,26.126,154.320
C01743=1084.403,352.158,406.265,176.617,26.131,154.321
C01744=1084.409,352.406,406.229,176.620,26.137,154.321
C01745=1084.416,352.653,406.194,176.623,26.142,154.322
C01746=1084.421,352.901,406.160,176.626,26.147,154.323
C01747=1084.427,353.149,406.124,176.630,26.152,154.324
C01748=1084.433,353.395,406.089,176.633,26.157,154.325
C01749=1084.439,353.643,406.053,176.636,26.163,154.326
C01750=1084.445,353.891,406.018,176.639,26.168,154.327
C01751=1084.451,354.138,405.984,176.642,26.173,154.327
C01752=1084.457,354.386,405.948,176.646,26.179,154.328
C01753=1084.463,354.633,405.912,176.648,26.184,154.329
C01754=1084.469,354.880,405.877,176.652,26.189,154.330
C01755=1084.475,355.128,405.842,176.655,26.194,154.331
C01756=1084.481,355.375,405.806,176.659,26.200,154.332
C01757=1084.486,355.623,405.771,176.661,26.205,154.333
C01758=1084.492,355.871,405.736,176.665,26.210,154.334
C01759=1084.498,356.117,405.701,176.668,26.216,154.335
C01760=1084.504,356.365,405.665,176.671,26.221,154.335
C01761=1084.510,356.613,405.629,176.674,26.227,154.336
C01762=1084.520,357.016,405.571,176.679,26.235,154.338
C01763=1084.531,357.420,405.513,176.684,26.244,154.339
C01764=1084.540,357.823,405.455,176.690,26.253,154.341
C01765=1084.550,358.227,405.397,176.695,26.262,154.342
C01766=1084.556,358.475,405.361,176.699,26.267,154.343
C01767=1084.563,358.722,405.326,176.702,26.273,154.344
C01768=1084.568,358.969,405.290,176.705,26.278,154.345
C01769=1084.574,359.216,405.254,176.708,26.283,154.346
C01770=1084.580,359.464,405.219,176.712,26.289,154.347
C01771=1084.586,359.712,405.183,176.715,26.294,154.348
C01772=1084.593,359.959,405.146,176.718,26.300,154.349
C01773=1084.598,360.206,405.111,176.721,26.306,154.350
C01774=1084.604,360.454,405.075,176.725,26.311,154.351
C01775=1084.610,360.701,405.040,176.727,26.317,154.351
C01776=1084.617,360.948,405.003,176.731,26.323,154.353
C01777=1084.622,361.195,404.968,176.734,26.328,154.353
C01778=1084.628,361.443,404.932,176.737,26.334,154.354
C01779=1084.634,361.690,404.896,176.740,26.339,154.355
C01780=1084.640,361.938,404.860,176.744,26.345,154.356
C01781=1084.647,362.185,404.823,176.747,26.350,154.357
C01782=1084.653,362.432,404.788,176.750,26.356,154.358
C01783=1084.658,362.679,404.752,176.753,26.362,154.359
C01784=1084.664,362.926,404.716,176.757,26.367,154.360
C01785=1084.671,363.173,404.679,176.759,26.373,154.361
C01786=1084.677,363.421,404.644,176.763,26.379,154.362
C01787=1084.683,363.668,404.607,176.766,26.384,154.363
C01788=1084.689,363.916,404.572,176.769,26.390,154.364
C01789=1084.696,364.163,404.535,176.772,26.395,154.365
C01790=1084.702,364.411,404.499,176.776,26.401,154.366
C01791=1084.708,364.658,404.463,176.779,26.407,154.367
C01792=1084.714,364.905,404.426,176.782,26.413,154.368
C01793=1084.719,365.152,404.391,176.786,26.419,154.369
C01794=1084.725,365.399,404.354,176.789,26.424,154.370
C01795=1084.732,365.646,404.318,176.792,26.430,154.371
C01796=1084.738,365.894,404.282,176.795,26.436,154.372
C01797=1084.743,366.141,404.245,176.798,26.442,154.373
C01798=1084.750,366.388,404.208,176.802,26.448,154.374
C01799=1084.756,366.635,404.172,176.805,26.453,154.375
C01800=1084.762,366.883,404.135,176.809,26.459,154.376
C01801=1084.768,367.130,404.099,176.811,26.465,154.377
C01802=1084.774,367.377,404.063,176.815,26.471,154.378
C01803=1084.780,367.624,404.026,176.818,26.477,154.379
C01804=1084.786,367.872,403.989,176.821,26.483,154.380
C01805=1084.792,368.119,403.953,176.825,26.489,154.381
C01806=1084.798,368.366,403.916,176.827,26.495,154.382
C01807=1084.804,368.613,403.879,176.831,26.501,154.383
C01808=1084.810,368.860,403.843,176.835,26.507,154.384
C01809=1084.816,369.108,403.806,176.837,26.513,154.386
C01810=1084.822,369.355,403.769,176.841,26.519,154.387
C01811=1084.829,369.602,403.733,176.844,26.525,154.388
C01812=1084.834,369.849,403.696,176.847,26.531,154.389
C01813=1084.841,370.096,403.660,176.851,26.537,154.390
C01814=1084.846,370.306,403.628,176.854,26.542,154.391
C01815=1084.850,370.516,403.598,176.857,26.547,154.392
C01816=1084.856,370.725,403.566,176.859,26.552,154.392
C01817=1084.861,370.935,403.535,176.862,26.558,154.393
C01818=1084.866,371.145,403.504,176.864,26.563,154.394
